KUKA KRL program: MyProgram_053().src

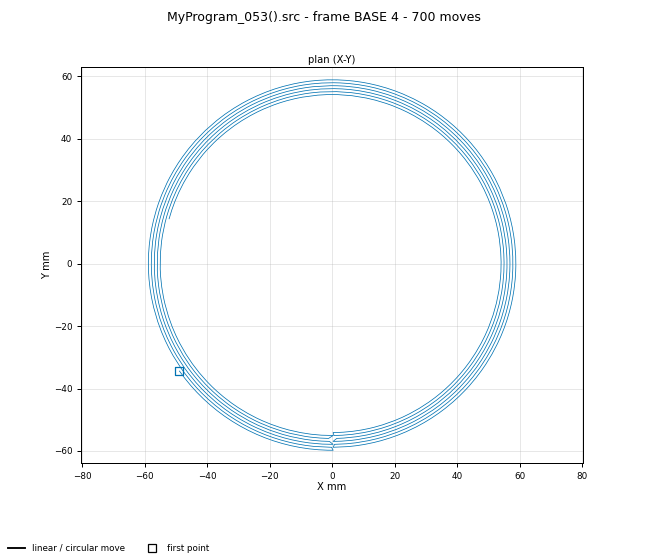
[picture p0: tool path of MyProgram_053().src in frame BASE 4, 700 of 700 moves have a stored position in this frame; points joined in program order, loops and branches not executed]
&ACCESS RVP
&REL 1
&PARAM TEMPLATE = C:\KRC\Roboter\Template\vorgabe
&PARAM EDITMASK = *
DEF MyProgram_053()
; ---- Setting reference (Base) ----
$BASE = BASE_DATA[4]

; --------------------------
; ---- Setting tool (TCP) ----
$TOOL = TOOL_DATA[3]
; --------------------------

$VEL.CP = VEL_APROX_PRINT
Startdeposition()
$VEL.CP = VEL_PRINT
LIN {X -48.8632,Y -34.4133,Z 68,A -149.9569,B 24.8869,C -2.4546,E1 24.8703,E2 233.9188} C_DIS
LIN {X -47.1157,Y -36.7695,Z 68,A -147.1292,B 24.8875,C -2.4482,E1 24.8751,E2 231.0929} C_DIS
LIN {X -45.2548,Y -39.0371,Z 68,A -144.3022,B 24.8881,C -2.4421,E1 24.8802,E2 228.2675} C_DIS
LIN {X -43.2848,Y -41.2106,Z 68,A -141.476,B 24.8886,C -2.4363,E1 24.8855,E2 225.4427} C_DIS
LIN {X -41.2106,Y -43.2848,Z 68,A -138.6504,B 24.8891,C -2.4308,E1 24.8912,E2 222.6185} C_DIS
LIN {X -39.0371,Y -45.2548,Z 68,A -135.8256,B 24.8896,C -2.4257,E1 24.8971,E2 219.7948} C_DIS
LIN {X -36.7695,Y -47.1157,Z 68,A -133.0016,B 24.89,C -2.4208,E1 24.9032,E2 216.9717} C_DIS
LIN {X -34.4133,Y -48.8632,Z 68,A -130.1785,B 24.8904,C -2.4164,E1 24.9096,E2 214.1495} C_DIS
LIN {X -31.9743,Y -50.4929,Z 68,A -127.3562,B 24.8908,C -2.4123,E1 24.9162,E2 211.3278} C_DIS
LIN {X -29.4582,Y -52.001,Z 68,A -124.535,B 24.8911,C -2.4085,E1 24.923,E2 208.5071} C_DIS
LIN {X -26.8711,Y -53.3838,Z 68,A -121.7145,B 24.8914,C -2.4052,E1 24.93,E2 205.6868} C_DIS
LIN {X -24.2194,Y -54.638,Z 68,A -118.8949,B 24.8917,C -2.4022,E1 24.9372,E2 202.8673} C_DIS
LIN {X -21.5092,Y -55.7606,Z 68,A -116.0763,B 24.8919,C -2.3996,E1 24.9445,E2 200.0486} C_DIS
LIN {X -18.7473,Y -56.7488,Z 68,A -113.2587,B 24.8921,C -2.3975,E1 24.9519,E2 197.2308} C_DIS
LIN {X -15.9402,Y -57.6003,Z 68,A -110.442,B 24.8923,C -2.3957,E1 24.9595,E2 194.4137} C_DIS
LIN {X -13.0946,Y -58.3131,Z 68,A -107.6262,B 24.8924,C -2.3943,E1 24.9672,E2 191.5974} C_DIS
LIN {X -10.2176,Y -58.8854,Z 68,A -104.8115,B 24.8925,C -2.3934,E1 24.9749,E2 188.7819} C_DIS
LIN {X -7.3159,Y -59.3158,Z 68,A -101.9978,B 24.8925,C -2.3929,E1 24.9827,E2 185.9674} C_DIS
LIN {X -4.3966,Y -59.6033,Z 68,A -99.185,B 24.8925,C -2.3928,E1 24.9905,E2 183.1534} C_DIS
LIN {X -1.4667,Y -59.7473,Z 68,A -96.3732,B 24.8925,C -2.3931,E1 24.9984,E2 180.3404} C_DIS
LIN {X 0.3491,Y -59.761,Z 68,A -94.9522,B 24.8931,C -2.3867,E1 25.0023,E2 178.9345} C_DIS
Enddeposition()
LIN {X 0.3491,Y -59.761,Z 68,A -94.9522,B 24.8931,C -2.3867,E1 25.0023,E2 178.9345} C_DIS
Startdeposition()
$VEL.CP = VEL_PRINT
LIN {X -0.1819,Y -58.8204,Z 68,A -97.1859,B 24.8948,C -2.3675,E1 24.9959,E2 181.214} C_DIS
LIN {X -5.9002,Y -58.5242,Z 68,A -102.0888,B 24.8936,C -2.3811,E1 24.9823,E2 186.0865} C_DIS
LIN {X -8.5559,Y -58.1955,Z 68,A -104.7263,B 24.8936,C -2.381,E1 24.975,E2 188.7262} C_DIS
LIN {X -11.2936,Y -57.7263,Z 68,A -107.3881,B 24.8935,C -2.3828,E1 24.9677,E2 191.3865} C_DIS
LIN {X -13.5936,Y -57.2291,Z 68,A -109.6463,B 24.8933,C -2.3845,E1 24.9616,E2 193.6434} C_DIS
LIN {X -16.2017,Y -56.5453,Z 68,A -112.2527,B 24.8931,C -2.3865,E1 24.9546,E2 196.2491} C_DIS
LIN {X -18.7885,Y -55.7389,Z 68,A -114.9287,B 24.8931,C -2.3878,E1 24.9475,E2 198.9269} C_DIS
LIN {X -21.2101,Y -54.8641,Z 68,A -117.4602,B 24.8928,C -2.3896,E1 24.9408,E2 201.4594} C_DIS
LIN {X -23.7558,Y -53.8105,Z 68,A -120.2317,B 24.8928,C -2.3907,E1 24.9337,E2 204.2348} C_DIS
LIN {X -25.9322,Y -52.7959,Z 68,A -122.5861,B 24.8925,C -2.3931,E1 24.9278,E2 206.5894} C_DIS
LIN {X -28.4573,Y -51.479,Z 68,A -125.2177,B 24.892,C -2.3994,E1 24.9213,E2 209.2134} C_DIS
LIN {X -30.7514,Y -50.1414,Z 68,A -127.767,B 24.8916,C -2.4038,E1 24.9152,E2 211.7601} C_DIS
LIN {X -32.928,Y -48.74,Z 68,A -130.3398,B 24.8913,C -2.4067,E1 24.9092,E2 214.3343} C_DIS
LIN {X -35.0695,Y -47.2236,Z 68,A -133.0589,B 24.8912,C -2.4079,E1 24.9031,E2 217.06} C_DIS
LIN {X -37.4099,Y -45.3916,Z 68,A -135.9134,B 24.8906,C -2.4139,E1 24.8968,E2 219.9109} C_DIS
LIN {X -39.5852,Y -43.5076,Z 68,A -138.9686,B 24.8906,C -2.4147,E1 24.8905,E2 222.9763} C_DIS
LIN {X -41.8366,Y -41.3466,Z 68,A -141.552,B 24.8892,C -2.4292,E1 24.8854,E2 225.536} C_DIS
LIN {X -43.5144,Y -39.5778,Z 68,A -144.139,B 24.8892,C -2.4305,E1 24.8804,E2 228.1313} C_DIS
LIN {X -45.2938,Y -37.5276,Z 68,A -146.7416,B 24.8885,C -2.4373,E1 24.8757,E2 230.7297} C_DIS
LIN {X -47.1481,Y -35.17,Z 68,A -149.431,B 24.8875,C -2.4483,E1 24.8712,E2 233.4055} C_DIS
LIN {X -48.4091,Y -33.4131,Z 68,A -151.8886,B 24.8875,C -2.4472,E1 24.8672,E2 235.8778} C_DIS
LIN {X -50.8588,Y -29.5512,Z 68,A -156.2944,B 24.8865,C -2.4595,E1 24.8607,E2 240.2766} C_DIS
LIN {X -52.1891,Y -27.1337,Z 68,A -159.076,B 24.886,C -2.4651,E1 24.857,E2 243.0598} C_DIS
LIN {X -53.4194,Y -24.6223,Z 68,A -161.8237,B 24.8853,C -2.4722,E1 24.8538,E2 245.8054} C_DIS
LIN {X -54.6088,Y -21.8592,Z 68,A -164.7604,B 24.8845,C -2.4803,E1 24.8506,E2 248.739} C_DIS
LIN {X -55.7868,Y -18.6465,Z 68,A -167.6273,B 24.8829,C -2.498,E1 24.8479,E2 251.5798} C_DIS
LIN {X -57.0985,Y -14.1292,Z 68,A -172.2395,B 24.8816,C -2.5111,E1 24.8444,E2 256.1874} C_DIS
LIN {X -57.7937,Y -10.9433,Z 68,A -175.929,B 24.8816,C -2.512,E1 24.8422,E2 259.8966} C_DIS
LIN {X -58.2622,Y -8.0862,Z 68,A -178.8137,B 24.8808,C -2.5196,E1 24.841,E2 262.7802} C_DIS
LIN {X -58.6196,Y -4.8584,Z 68,A 178.0495,B 24.8799,C -2.5299,E1 24.8402,E2 265.9112} C_DIS
LIN {X -58.7827,Y -2.13,Z 68,A 175.3754,B 24.8791,C -2.538,E1 24.8398,E2 268.582} C_DIS
LIN {X -58.82,Y 0.4129,Z 68,A 172.7179,B 24.8786,C -2.5428,E1 24.8398,E2 271.2441} C_DIS
LIN {X -58.7265,Y 3.3237,Z 68,A 170.0395,B 24.8775,C -2.5544,E1 24.8401,E2 273.9108} C_DIS
LIN {X -58.5256,Y 5.8861,Z 68,A 167.6002,B 24.8766,C -2.5634,E1 24.8408,E2 276.3433} C_DIS
LIN {X -58.2079,Y 8.4688,Z 68,A 164.903,B 24.8761,C -2.5687,E1 24.8418,E2 279.044} C_DIS
LIN {X -57.7129,Y 11.3629,Z 68,A 162.0961,B 24.8752,C -2.5785,E1 24.8432,E2 281.844} C_DIS
LIN {X -57.1771,Y 13.8072,Z 68,A 159.7574,B 24.8743,C -2.5878,E1 24.8446,E2 284.1743} C_DIS
LIN {X -56.2843,Y 17.0892,Z 68,A 156.5483,B 24.8731,C -2.5998,E1 24.847,E2 287.3733} C_DIS
LIN {X -55.6014,Y 19.1939,Z 68,A 154.0471,B 24.8731,C -2.6005,E1 24.8493,E2 289.8871} C_DIS
LIN {X -54.5799,Y 21.9303,Z 68,A 150.4175,B 24.8735,C -2.5959,E1 24.853,E2 293.5481} C_DIS
LIN {X -52.8589,Y 25.805,Z 68,A 147.4075,B 24.8704,C -2.6269,E1 24.8565,E2 296.5002} C_DIS
LIN {X -52.0364,Y 27.4235,Z 68,A 145.281,B 24.8705,C -2.6259,E1 24.8592,E2 298.6405} C_DIS
LIN {X -50.7407,Y 29.7534,Z 68,A 142.7868,B 24.8696,C -2.635,E1 24.8627,E2 301.1259} C_DIS
LIN {X -49.2458,Y 32.1676,Z 68,A 139.8519,B 24.8692,C -2.6398,E1 24.8671,E2 304.0643} C_DIS
LIN {X -47.8916,Y 34.1501,Z 68,A 137.5081,B 24.8685,C -2.646,E1 24.8708,E2 306.4049} C_DIS
LIN {X -45.9649,Y 36.7021,Z 68,A 134.4363,B 24.8676,C -2.6549,E1 24.8761,E2 309.47} C_DIS
LIN {X -43.8935,Y 39.1557,Z 68,A 130.9326,B 24.8676,C -2.6562,E1 24.8825,E2 312.9864} C_DIS
LIN {X -40.5775,Y 42.5843,Z 68,A 126.1334,B 24.8667,C -2.6645,E1 24.892,E2 317.7861} C_DIS
LIN {X -36.8982,Y 45.8082,Z 68,A 121.4315,B 24.8655,C -2.676,E1 24.902,E2 322.4785} C_DIS
LIN {X -34.2453,Y 47.8237,Z 68,A 118.3432,B 24.8646,C -2.6854,E1 24.909,E2 325.5554} C_DIS
LIN {X -31.4406,Y 49.7134,Z 68,A 115.1794,B 24.8637,C -2.6939,E1 24.9163,E2 328.7091} C_DIS
LIN {X -28.7227,Y 51.3307,Z 68,A 112.2925,B 24.8628,C -2.7029,E1 24.9233,E2 331.5834} C_DIS
LIN {X -26.8061,Y 52.3571,Z 68,A 109.9748,B 24.8628,C -2.7027,E1 24.929,E2 333.9079} C_DIS
LIN {X -24.1417,Y 53.6378,Z 68,A 106.9814,B 24.8626,C -2.7049,E1 24.9366,E2 336.9034} C_DIS
LIN {X -21.1328,Y 54.894,Z 68,A 103.9362,B 24.8619,C -2.7116,E1 24.9445,E2 339.9394} C_DIS
LIN {X -18.4448,Y 55.8547,Z 68,A 101.1212,B 24.8616,C -2.7143,E1 24.9519,E2 342.7533} C_DIS
LIN {X -15.7595,Y 56.6706,Z 68,A 98.3718,B 24.8614,C -2.7169,E1 24.9593,E2 345.5009} C_DIS
LIN {X -12.2609,Y 57.529,Z 68,A 95.0311,B 24.8607,C -2.7233,E1 24.9683,E2 348.8308} C_DIS
LIN {X -9.8349,Y 57.9925,Z 68,A 92.5949,B 24.8606,C -2.7246,E1 24.975,E2 351.2667} C_DIS
LIN {X -7.116,Y 58.389,Z 68,A 89.8714,B 24.8606,C -2.7253,E1 24.9826,E2 353.9905} C_DIS
LIN {X -4.5936,Y 58.6408,Z 68,A 87.3044,B 24.8606,C -2.7246,E1 24.9897,E2 356.5605} C_DIS
LIN {X -1.5185,Y 58.8015,Z 68,A 84.2474,B 24.8606,C -2.7244,E1 24.9982,E2 359.6185} C_DIS
LIN {X 1.6458,Y 58.7976,Z 68,A 81.222,B 24.8604,C -2.726,E1 25.0067,E2 362.6398} C_DIS
LIN {X 4.5596,Y 58.6435,Z 68,A 78.5253,B 24.8601,C -2.7289,E1 25.0142,E2 365.3284} C_DIS
LIN {X 7.0083,Y 58.4016,Z 68,A 76.0735,B 24.8603,C -2.7274,E1 25.021,E2 367.782} C_DIS
LIN {X 9.7413,Y 58.0082,Z 68,A 73.563,B 24.86,C -2.7303,E1 25.0279,E2 370.2833} C_DIS
LIN {X 11.8943,Y 57.6053,Z 68,A 71.2881,B 24.8604,C -2.7265,E1 25.0341,E2 372.5645} C_DIS
LIN {X 14.4994,Y 57.0055,Z 68,A 68.5573,B 24.8608,C -2.7225,E1 25.0416,E2 375.3009} C_DIS
LIN {X 17.4989,Y 56.1572,Z 68,A 65.5349,B 24.861,C -2.7206,E1 25.0496,E2 378.3225} C_DIS
LIN {X 20.1878,Y 55.2475,Z 68,A 62.629,B 24.8615,C -2.7153,E1 25.0573,E2 381.2352} C_DIS
LIN {X 22.6593,Y 54.2811,Z 68,A 59.8471,B 24.8622,C -2.7085,E1 25.0645,E2 384.0268} C_DIS
LIN {X 26.0847,Y 52.7203,Z 68,A 56.5042,B 24.862,C -2.7111,E1 25.0729,E2 387.3549} C_DIS
LIN {X 29.0426,Y 51.1513,Z 68,A 53.5864,B 24.8617,C -2.7141,E1 25.08,E2 390.2571} C_DIS
LIN {X 30.8083,Y 50.1077,Z 68,A 51.3127,B 24.8626,C -2.7052,E1 25.0855,E2 392.5448} C_DIS
LIN {X 32.9546,Y 48.722,Z 68,A 49.0436,B 24.8625,C -2.7061,E1 25.0908,E2 394.8043} C_DIS
LIN {X 34.8992,Y 47.3489,Z 68,A 46.4804,B 24.8634,C -2.6968,E1 25.0966,E2 397.3804} C_DIS
LIN {X 37.2606,Y 45.5144,Z 68,A 43.5291,B 24.864,C -2.6907,E1 25.1031,E2 400.3352} C_DIS
LIN {X 39.066,Y 43.9743,Z 68,A 41.4039,B 24.864,C -2.6904,E1 25.1075,E2 402.4528} C_DIS
LIN {X 41.0256,Y 42.1523,Z 68,A 38.6909,B 24.8648,C -2.6827,E1 25.113,E2 405.1728} C_DIS
LIN {X 42.9045,Y 40.2373,Z 68,A 36.1779,B 24.8652,C -2.6794,E1 25.1179,E2 407.6827} C_DIS
LIN {X 44.4749,Y 38.4953,Z 68,A 33.8185,B 24.8659,C -2.6726,E1 25.1222,E2 410.0477} C_DIS
LIN {X 46.2369,Y 36.3594,Z 68,A 31.1846,B 24.8664,C -2.6678,E1 25.1268,E2 412.6808} C_DIS
LIN {X 47.8292,Y 34.2376,Z 68,A 28.6547,B 24.8669,C -2.6627,E1 25.131,E2 415.2104} C_DIS
LIN {X 49.4968,Y 31.7789,Z 68,A 25.6809,B 24.8678,C -2.6536,E1 25.1356,E2 418.1909} C_DIS
LIN {X 51.014,Y 29.2815,Z 68,A 22.9579,B 24.8682,C -2.649,E1 25.1395,E2 420.9109} C_DIS
LIN {X 52.2323,Y 27.0503,Z 68,A 19.8319,B 24.8704,C -2.6275,E1 25.1436,E2 424.0712} C_DIS
LIN {X 53.6588,Y 24.0952,Z 68,A 16.7232,B 24.8711,C -2.6206,E1 25.1472,E2 427.1794} C_DIS
LIN {X 55.5872,Y 19.2344,Z 68,A 12.4414,B 24.8707,C -2.6247,E1 25.1514,E2 431.4277} C_DIS
LIN {X 56.2835,Y 17.0915,Z 68,A 9.9975,B 24.8719,C -2.6124,E1 25.1535,E2 433.8867} C_DIS
LIN {X 57.0667,Y 14.2598,Z 68,A 7.2199,B 24.8725,C -2.6058,E1 25.1554,E2 436.6639} C_DIS
LIN {X 57.6695,Y 11.5813,Z 68,A 4.5156,B 24.8734,C -2.597,E1 25.157,E2 439.3734} C_DIS
LIN {X 58.1359,Y 8.9473,Z 68,A 1.9962,B 24.874,C -2.591,E1 25.1582,E2 441.8921} C_DIS
LIN {X 58.4681,Y 6.4352,Z 68,A -0.6025,B 24.875,C -2.5803,E1 25.159,E2 444.5008} C_DIS
LIN {X 58.7635,Y 2.5865,Z 68,A -4.6079,B 24.8767,C -2.5628,E1 25.1597,E2 448.5238} C_DIS
LIN {X 58.8186,Y -0.5568,Z 68,A -7.0159,B 24.8762,C -2.5684,E1 25.1597,E2 450.9042} C_DIS
LIN {X 58.7666,Y -2.5145,Z 68,A -9.2638,B 24.8775,C -2.5544,E1 25.1595,E2 453.1719} C_DIS
LIN {X 58.6012,Y -5.0835,Z 68,A -11.8045,B 24.8783,C -2.5457,E1 25.159,E2 455.718} C_DIS
LIN {X 58.2064,Y -8.479,Z 68,A -14.7537,B 24.8785,C -2.5441,E1 25.1579,E2 458.6535} C_DIS
LIN {X 57.7979,Y -10.9214,Z 68,A -17.1892,B 24.8793,C -2.536,E1 25.1568,E2 461.094} C_DIS
LIN {X 57.378,Y -12.9497,Z 68,A -19.3393,B 24.8802,C -2.5265,E1 25.1555,E2 463.2539} C_DIS
LIN {X 56.7813,Y -15.3532,Z 68,A -21.7826,B 24.881,C -2.5183,E1 25.1538,E2 465.7025} C_DIS
LIN {X 55.9859,Y -18.0394,Z 68,A -24.5467,B 24.8818,C -2.5091,E1 25.1515,E2 468.4728} C_DIS
LIN {X 55.1025,Y -20.5821,Z 68,A -27.008,B 24.8822,C -2.5049,E1 25.1492,E2 470.9302} C_DIS
LIN {X 54.1298,Y -23.0182,Z 68,A -29.6221,B 24.8831,C -2.4958,E1 25.1464,E2 473.5513} C_DIS
LIN {X 52.9555,Y -25.6042,Z 68,A -32.7817,B 24.8847,C -2.4785,E1 25.1426,E2 476.7347} C_DIS
LIN {X 51.1574,Y -29.0321,Z 68,A -36.2551,B 24.8851,C -2.4745,E1 25.1379,E2 480.1994} C_DIS
LIN {X 49.1785,Y -32.2697,Z 68,A -39.6052,B 24.8853,C -2.4722,E1 25.133,E2 483.5379} C_DIS
LIN {X 47.8134,Y -34.2598,Z 68,A -42.1617,B 24.8863,C -2.4611,E1 25.1289,E2 486.1083} C_DIS
LIN {X 46.0279,Y -36.6239,Z 68,A -45.2761,B 24.8875,C -2.4483,E1 25.1235,E2 489.2384} C_DIS
LIN {X 43.9528,Y -39.09,Z 68,A -47.6687,B 24.8867,C -2.4574,E1 25.1192,E2 491.5985} C_DIS
LIN {X 42.6761,Y -40.4803,Z 68,A -49.9852,B 24.8881,C -2.442,E1 25.1148,E2 493.9414} C_DIS
LIN {X 40.7579,Y -42.4104,Z 68,A -52.5538,B 24.8885,C -2.4375,E1 25.1096,E2 496.5096} C_DIS
LIN {X 38.7295,Y -44.2704,Z 68,A -55.3493,B 24.8893,C -2.4288,E1 25.1038,E2 499.3146} C_DIS
LIN {X 36.2424,Y -46.3294,Z 68,A -58.2487,B 24.8894,C -2.4276,E1 25.0975,E2 502.2061} C_DIS
LIN {X 34.2378,Y -47.829,Z 68,A -60.8411,B 24.8902,C -2.4191,E1 25.0917,E2 504.8092} C_DIS
LIN {X 31.8563,Y -49.4472,Z 68,A -63.6213,B 24.8906,C -2.4143,E1 25.0852,E2 507.5917} C_DIS
LIN {X 29.4736,Y -50.9037,Z 68,A -66.3447,B 24.8911,C -2.4093,E1 25.0786,E2 510.3185} C_DIS
LIN {X 26.9019,Y -52.3082,Z 68,A -69.5131,B 24.8921,C -2.3976,E1 25.0708,E2 513.5057} C_DIS
LIN {X 23.6635,Y -53.8508,Z 68,A -72.6989,B 24.892,C -2.399,E1 25.0627,E2 516.6802} C_DIS
LIN {X 21.0515,Y -54.9247,Z 68,A -75.3162,B 24.892,C -2.3981,E1 25.0559,E2 519.2936} C_DIS
LIN {X 18.5531,Y -55.8175,Z 68,A -77.9819,B 24.8925,C -2.3931,E1 25.0489,E2 521.9659} C_DIS
LIN {X 15.6483,Y -56.7016,Z 68,A -80.8451,B 24.8926,C -2.3919,E1 25.0412,E2 524.8271} C_DIS
LIN {X 13.3649,Y -57.2821,Z 68,A -83.2555,B 24.8931,C -2.3872,E1 25.0346,E2 527.2451} C_DIS
LIN {X 10.4333,Y -57.8877,Z 68,A -86.3232,B 24.8936,C -2.3816,E1 25.0262,E2 530.3225} C_DIS
LIN {X 7.9324,Y -58.2841,Z 68,A -88.6588,B 24.8935,C -2.3827,E1 25.0198,E2 532.6536} C_DIS
LIN {X 5.1225,Y -58.5975,Z 68,A -91.9162,B 24.8945,C -2.3708,E1 25.0106,E2 535.9372} C_DIS
LIN {X 0.3303,Y -58.8102,Z 68,A -94.5805,B 24.8909,C -2.4111,E1 25.0035,E2 538.505} C_DIS
Enddeposition()
LIN {X 0.3303,Y -58.8102,Z 68,A -94.5805,B 24.8909,C -2.4111,E1 25.0035,E2 538.505} C_DIS
Startdeposition()
$VEL.CP = VEL_PRINT
LIN {X 0.78,Y -57.8714,Z 68,A -94.0127,B 24.8892,C -2.4297,E1 25.0052,E2 537.8931} C_DIS
LIN {X 4.6739,Y -57.6876,Z 68,A -90.3787,B 24.8895,C -2.4267,E1 25.0153,E2 534.2679} C_DIS
LIN {X 7.6047,Y -57.3751,Z 68,A -87.8197,B 24.89,C -2.4209,E1 25.0223,E2 531.7245} C_DIS
LIN {X 11.7052,Y -56.6807,Z 68,A -83.3977,B 24.8891,C -2.4305,E1 25.0346,E2 527.2844} C_DIS
LIN {X 14.3445,Y -56.0709,Z 68,A -80.677,B 24.8888,C -2.434,E1 25.0419,E2 524.5596} C_DIS
LIN {X 16.8623,Y -55.3665,Z 68,A -77.3217,B 24.887,C -2.4535,E1 25.051,E2 521.1637} C_DIS
LIN {X 20.8071,Y -54.0081,Z 68,A -74.1057,B 24.8884,C -2.4389,E1 25.0593,E2 517.9892} C_DIS
LIN {X 23.7341,Y -52.7864,Z 68,A -71.0499,B 24.8881,C -2.4416,E1 25.0672,E2 514.9342} C_DIS
LIN {X 26.6333,Y -51.3855,Z 68,A -67.275,B 24.8864,C -2.4598,E1 25.0767,E2 511.1266} C_DIS
LIN {X 29.9387,Y -49.5318,Z 68,A -63.9811,B 24.8868,C -2.4562,E1 25.0846,E2 507.8509} C_DIS
LIN {X 32.2718,Y -48.0446,Z 68,A -61.2572,B 24.8863,C -2.4611,E1 25.0909,E2 505.1244} C_DIS
LIN {X 34.2385,Y -46.663,Z 68,A -58.3006,B 24.8846,C -2.4791,E1 25.0977,E2 502.1358} C_DIS
LIN {X 37.217,Y -44.3246,Z 68,A -54.7007,B 24.8842,C -2.4838,E1 25.1055,E2 498.5384} C_DIS
LIN {X 39.9475,Y -41.8807,Z 68,A -51.5822,B 24.8845,C -2.4805,E1 25.1118,E2 495.4403} C_DIS
LIN {X 41.9102,Y -39.9168,Z 68,A -49.1055,B 24.8845,C -2.4809,E1 25.1166,E2 492.9733} C_DIS
LIN {X 43.3694,Y -38.325,Z 68,A -46.807,B 24.8836,C -2.49,E1 25.1209,E2 490.6637} C_DIS
LIN {X 45.094,Y -36.2803,Z 68,A -43.6872,B 24.882,C -2.5077,E1 25.1265,E2 487.5162} C_DIS
LIN {X 47.3207,Y -33.3254,Z 68,A -40.5794,B 24.8822,C -2.5046,E1 25.1316,E2 484.4308} C_DIS
LIN {X 49.4641,Y -30.0499,Z 68,A -36.7413,B 24.8813,C -2.5145,E1 25.1374,E2 480.5885} C_DIS
LIN {X 51.079,Y -27.2161,Z 68,A -33.062,B 24.8794,C -2.5343,E1 25.1424,E2 476.8817} C_DIS
LIN {X 52.4942,Y -24.3734,Z 68,A -29.8313,B 24.8784,C -2.5456,E1 25.1463,E2 473.6416} C_DIS
LIN {X 53.9012,Y -21.0802,Z 68,A -26.7204,B 24.8784,C -2.546,E1 25.1495,E2 470.5469} C_DIS
LIN {X 54.8699,Y -18.412,Z 68,A -23.9576,B 24.8776,C -2.5535,E1 25.1521,E2 467.782} C_DIS
LIN {X 55.6901,Y -15.7582,Z 68,A -21.1575,B 24.8767,C -2.5632,E1 25.1543,E2 464.975} C_DIS
LIN {X 56.3798,Y -13.0776,Z 68,A -18.2243,B 24.8754,C -2.5763,E1 25.1562,E2 462.0278} C_DIS
LIN {X 57.06,Y -9.6894,Z 68,A -15.5141,B 24.876,C -2.5703,E1 25.1576,E2 459.3477} C_DIS
LIN {X 57.3952,Y -7.4494,Z 68,A -12.8681,B 24.8744,C -2.5868,E1 25.1587,E2 456.6781} C_DIS
LIN {X 57.6691,Y -4.9056,Z 68,A -10.2228,B 24.8733,C -2.5975,E1 25.1594,E2 454.0233} C_DIS
LIN {X 57.8559,Y -1.5642,Z 68,A -7.0469,B 24.8726,C -2.6047,E1 25.1598,E2 450.8492} C_DIS
LIN {X 57.835,Y 2.208,Z 68,A -2.7929,B 24.8702,C -2.6287,E1 25.1595,E2 446.5637} C_DIS
LIN {X 57.5655,Y 5.9934,Z 68,A 0.3996,B 24.8704,C -2.6272,E1 25.1587,E2 443.3939} C_DIS
LIN {X 57.306,Y 8.1072,Z 68,A 2.4235,B 24.87,C -2.6317,E1 25.158,E2 441.3712} C_DIS
LIN {X 56.8276,Y 10.9692,Z 68,A 5.2758,B 24.8691,C -2.64,E1 25.1566,E2 438.5158} C_DIS
LIN {X 56.281,Y 13.4982,Z 68,A 7.9804,B 24.868,C -2.6511,E1 25.1549,E2 435.8006} C_DIS
LIN {X 55.5222,Y 16.3404,Z 68,A 11.1766,B 24.8665,C -2.6665,E1 25.1524,E2 432.5866} C_DIS
LIN {X 54.66,Y 19.0265,Z 68,A 13.9132,B 24.8658,C -2.6733,E1 25.1499,E2 429.8492} C_DIS
LIN {X 53.2238,Y 22.7362,Z 68,A 17.4466,B 24.8656,C -2.6751,E1 25.1462,E2 426.3311} C_DIS
LIN {X 52.3711,Y 24.6379,Z 68,A 19.8863,B 24.8642,C -2.6895,E1 25.1433,E2 423.8704} C_DIS
LIN {X 50.7121,Y 27.8945,Z 68,A 23.1418,B 24.864,C -2.6908,E1 25.1391,E2 420.629} C_DIS
LIN {X 49.2661,Y 30.3755,Z 68,A 25.9891,B 24.8633,C -2.6983,E1 25.135,E2 417.7785} C_DIS
LIN {X 46.9666,Y 33.8217,Z 68,A 30.0766,B 24.8623,C -2.7082,E1 25.1285,E2 413.6878} C_DIS
LIN {X 45.1647,Y 36.1933,Z 68,A 32.9551,B 24.8617,C -2.7136,E1 25.1236,E2 410.8102} C_DIS
LIN {X 42.987,Y 38.7539,Z 68,A 36.4163,B 24.8606,C -2.724,E1 25.1172,E2 407.3397} C_DIS
LIN {X 40.9213,Y 40.9299,Z 68,A 39.2019,B 24.8604,C -2.7262,E1 25.1118,E2 404.561} C_DIS
LIN {X 38.9759,Y 42.7858,Z 68,A 42.0048,B 24.8595,C -2.7346,E1 25.1061,E2 401.7494} C_DIS
LIN {X 35.9351,Y 45.3693,Z 68,A 45.8643,B 24.859,C -2.7399,E1 25.0977,E2 397.8922} C_DIS
LIN {X 33.3247,Y 47.3211,Z 68,A 49.4908,B 24.8575,C -2.7541,E1 25.0895,E2 394.2447} C_DIS
LIN {X 30.0673,Y 49.4536,Z 68,A 52.826,B 24.8581,C -2.7487,E1 25.0817,E2 390.9332} C_DIS
LIN {X 28.3743,Y 50.4444,Z 68,A 54.9276,B 24.8575,C -2.7548,E1 25.0765,E2 388.8234} C_DIS
LIN {X 25.8658,Y 51.7755,Z 68,A 57.6285,B 24.8573,C -2.756,E1 25.0698,E2 386.1271} C_DIS
LIN {X 23.1034,Y 53.0654,Z 68,A 60.6915,B 24.8569,C -2.7603,E1 25.062,E2 383.0614} C_DIS
LIN {X 19.916,Y 54.3417,Z 68,A 64.0369,B 24.8567,C -2.7624,E1 25.0533,E2 379.7183} C_DIS
LIN {X 17.1237,Y 55.2855,Z 68,A 67.2148,B 24.8559,C -2.7701,E1 25.0449,E2 376.528} C_DIS
LIN {X 13.9518,Y 56.1703,Z 68,A 70.152,B 24.8564,C -2.7654,E1 25.037,E2 373.6067} C_DIS
LIN {X 11.4099,Y 56.7413,Z 68,A 72.7812,B 24.8561,C -2.7676,E1 25.0298,E2 370.9756} C_DIS
LIN {X 8.4584,Y 57.2558,Z 68,A 75.9579,B 24.8556,C -2.7728,E1 25.021,E2 367.7895} C_DIS
LIN {X 5.2145,Y 57.6413,Z 68,A 78.8815,B 24.8562,C -2.767,E1 25.0129,E2 364.8818} C_DIS
LIN {X 2.545,Y 57.8207,Z 68,A 81.3542,B 24.8566,C -2.7634,E1 25.0061,E2 362.4185} C_DIS
LIN {X 0.4353,Y 57.875,Z 68,A 83.7312,B 24.856,C -2.7688,E1 24.9994,E2 360.0289} C_DIS
LIN {X -3.3089,Y 57.7821,Z 68,A 87.6438,B 24.8557,C -2.7717,E1 24.9884,E2 356.1087} C_DIS
LIN {X -6.6039,Y 57.4988,Z 68,A 90.5962,B 24.8565,C -2.7638,E1 24.9803,E2 353.1736} C_DIS
LIN {X -9.1846,Y 57.1442,Z 68,A 93.2568,B 24.8565,C -2.7636,E1 24.9729,E2 350.5111} C_DIS
LIN {X -11.1973,Y 56.7837,Z 68,A 95.4579,B 24.8564,C -2.7655,E1 24.9669,E2 348.3032} C_DIS
LIN {X -14.0822,Y 56.1382,Z 68,A 98.1948,B 24.857,C -2.7591,E1 24.9595,E2 345.5776} C_DIS
LIN {X -16.899,Y 55.3551,Z 68,A 101.1648,B 24.8572,C -2.7575,E1 24.9515,E2 342.6067} C_DIS
LIN {X -19.5753,Y 54.4664,Z 68,A 103.8788,B 24.8577,C -2.7526,E1 24.9444,E2 339.8991} C_DIS
LIN {X -22.3538,Y 53.3856,Z 68,A 106.9839,B 24.8578,C -2.7515,E1 24.9363,E2 336.7897} C_DIS
LIN {X -25.3527,Y 52.0293,Z 68,A 110.1218,B 24.8585,C -2.7443,E1 24.9284,E2 333.6611} C_DIS
LIN {X -27.4671,Y 50.944,Z 68,A 113.0058,B 24.8579,C -2.7503,E1 24.9212,E2 330.7548} C_DIS
LIN {X -30.3801,Y 49.2631,Z 68,A 115.7209,B 24.8597,C -2.7331,E1 24.9148,E2 328.0726} C_DIS
LIN {X -32.9008,Y 47.6158,Z 68,A 118.8661,B 24.86,C -2.7303,E1 24.9075,E2 324.9234} C_DIS
LIN {X -34.952,Y 46.131,Z 68,A 121.649,B 24.86,C -2.7303,E1 24.9013,E2 322.1309} C_DIS
LIN {X -38.0309,Y 43.6274,Z 68,A 125.0474,B 24.8618,C -2.7122,E1 24.894,E2 318.7624} C_DIS
LIN {X -39.9503,Y 41.878,Z 68,A 128.078,B 24.8616,C -2.7145,E1 24.8878,E2 315.7141} C_DIS
LIN {X -41.6921,Y 40.1432,Z 68,A 130.066,B 24.863,C -2.7008,E1 24.884,E2 313.7502} C_DIS
LIN {X -43.2066,Y 38.5086,Z 68,A 132.5738,B 24.863,C -2.7007,E1 24.8792,E2 311.2317} C_DIS
LIN {X -44.8223,Y 36.6158,Z 68,A 134.9729,B 24.8638,C -2.6933,E1 24.875,E2 308.8392} C_DIS
LIN {X -46.7908,Y 34.0639,Z 68,A 138.0557,B 24.8648,C -2.683,E1 24.8698,E2 305.7661} C_DIS
LIN {X -48.0905,Y 32.2039,Z 68,A 140.8524,B 24.8645,C -2.6864,E1 24.8654,E2 302.9474} C_DIS
LIN {X -49.9727,Y 29.1979,Z 68,A 144.0823,B 24.866,C -2.6717,E1 24.8607,E2 299.736} C_DIS
LIN {X -51.3637,Y 26.6755,Z 68,A 146.8569,B 24.8669,C -2.6622,E1 24.8571,E2 296.9694} C_DIS
LIN {X -52.8218,Y 23.6552,Z 68,A 150.0844,B 24.868,C -2.6509,E1 24.8533,E2 293.7513} C_DIS
LIN {X -53.6201,Y 21.785,Z 68,A 152.3867,B 24.8682,C -2.6498,E1 24.8508,E2 291.4388} C_DIS
LIN {X -54.7886,Y 18.6532,Z 68,A 155.5045,B 24.8695,C -2.6365,E1 24.8479,E2 288.3352} C_DIS
LIN {X -55.3682,Y 16.8536,Z 68,A 158.1009,B 24.8688,C -2.6432,E1 24.8457,E2 285.7079} C_DIS
LIN {X -56.4794,Y 12.6446,Z 68,A 161.8983,B 24.871,C -2.621,E1 24.8432,E2 281.9414} C_DIS
LIN {X -57.0063,Y 10.0022,Z 68,A 164.5573,B 24.8719,C -2.6125,E1 24.8419,E2 279.2869} C_DIS
LIN {X -57.4397,Y 7.1061,Z 68,A 167.4696,B 24.8727,C -2.6036,E1 24.8408,E2 276.3785} C_DIS
LIN {X -57.7841,Y 3.272,Z 68,A 171.0504,B 24.8743,C -2.5877,E1 24.84,E2 272.8142} C_DIS
LIN {X -57.876,Y -0.4305,Z 68,A 175.0736,B 24.8748,C -2.5822,E1 24.8398,E2 268.78} C_DIS
LIN {X -57.7878,Y -3.2048,Z 68,A 177.7218,B 24.8758,C -2.5719,E1 24.8401,E2 266.1406} C_DIS
LIN {X -57.4786,Y -6.776,Z 68,A -178.1855,B 24.876,C -2.5701,E1 24.8413,E2 262.0275} C_DIS
LIN {X -56.8854,Y -10.6693,Z 68,A -174.7203,B 24.8779,C -2.5507,E1 24.8429,E2 258.5881} C_DIS
LIN {X -56.3281,Y -13.3014,Z 68,A -171.1865,B 24.8772,C -2.5577,E1 24.8452,E2 255.0169} C_DIS
LIN {X -55.1745,Y -17.4811,Z 68,A -167.1306,B 24.8788,C -2.5409,E1 24.8485,E2 250.9778} C_DIS
LIN {X -53.8888,Y -21.1118,Z 68,A -164.0836,B 24.8811,C -2.5166,E1 24.8514,E2 247.9717} C_DIS
LIN {X -52.8045,Y -23.6939,Z 68,A -161.0594,B 24.8814,C -2.5132,E1 24.8548,E2 244.9389} C_DIS
LIN {X -51.5463,Y -26.3188,Z 68,A -158.1799,B 24.8822,C -2.5053,E1 24.8583,E2 242.0627} C_DIS
LIN {X -50.6502,Y -28.0057,Z 68,A -156.3925,B 24.8828,C -2.4984,E1 24.8607,E2 240.2823} C_DIS
LIN {X -49.7083,Y -29.6449,Z 68,A -154.0153,B 24.8824,C -2.5025,E1 24.8641,E2 237.883} C_DIS
LIN {X -47.1531,Y -33.5603,Z 68,A -150.0117,B 24.8846,C -2.4799,E1 24.8703,E2 233.9136} C_DIS
LIN {X -45.9103,Y -35.2414,Z 68,A -147.539,B 24.8844,C -2.4821,E1 24.8745,E2 231.4237} C_DIS
LIN {X -43.5847,Y -38.0799,Z 68,A -144.0307,B 24.8853,C -2.4716,E1 24.8808,E2 227.9243} C_DIS
LIN {X -41.6382,Y -40.1991,Z 68,A -141.1778,B 24.8859,C -2.4656,E1 24.8863,E2 225.0734} C_DIS
LIN {X -39.9557,Y -41.8728,Z 68,A -138.6526,B 24.886,C -2.464,E1 24.8913,E2 222.5414} C_DIS
LIN {X -37.1147,Y -44.4098,Z 68,A -135.5205,B 24.8878,C -2.4451,E1 24.8979,E2 219.4421} C_DIS
LIN {X -34.303,Y -46.6157,Z 68,A -131.4108,B 24.8874,C -2.4495,E1 24.907,E2 215.307} C_DIS
LIN {X -32.0434,Y -48.1973,Z 68,A -128.7427,B 24.8879,C -2.444,E1 24.9131,E2 212.6431} C_DIS
LIN {X -29.2489,Y -49.9417,Z 68,A -125.3329,B 24.8881,C -2.4421,E1 24.9213,E2 209.2272} C_DIS
LIN {X -26.2122,Y -51.6008,Z 68,A -122.1193,B 24.8888,C -2.4337,E1 24.9292,E2 206.0248} C_DIS
LIN {X -24.455,Y -52.4562,Z 68,A -119.7543,B 24.8883,C -2.4398,E1 24.9352,E2 203.6393} C_DIS
LIN {X -21.2149,Y -53.8482,Z 68,A -116.5985,B 24.8892,C -2.4298,E1 24.9433,E2 200.5002} C_DIS
LIN {X -18.1455,Y -54.9595,Z 68,A -113.2706,B 24.8892,C -2.429,E1 24.9521,E2 197.1677} C_DIS
LIN {X -15.2826,Y -55.8228,Z 68,A -110.3222,B 24.8895,C -2.4268,E1 24.96,E2 194.2197} C_DIS
LIN {X -12.8848,Y -56.4243,Z 68,A -107.8951,B 24.8896,C -2.4252,E1 24.9666,E2 191.7931} C_DIS
LIN {X -9.7967,Y -57.042,Z 68,A -104.8882,B 24.8899,C -2.4219,E1 24.9749,E2 188.791} C_DIS
LIN {X -7.2781,Y -57.4174,Z 68,A -102.2579,B 24.8898,C -2.4236,E1 24.9822,E2 186.1546} C_DIS
LIN {X -3.1822,Y -57.7891,Z 68,A -97.8455,B 24.8891,C -2.4305,E1 24.9945,E2 181.724} C_DIS
LIN {X 0.3229,Y -57.875,Z 68,A -95.2638,B 24.8907,C -2.4129,E1 25.0016,E2 179.184} C_DIS
Enddeposition()
LIN {X 0.3229,Y -57.875,Z 68,A -95.2638,B 24.8907,C -2.4129,E1 25.0016,E2 179.184} C_DIS
Startdeposition()
$VEL.CP = VEL_PRINT
LIN {X -0.8687,Y -56.9265,Z 68,A -97.0968,B 24.8904,C -2.4162,E1 24.9965,E2 181.009} C_DIS
LIN {X -3.413,Y -56.8303,Z 68,A -100.1238,B 24.8913,C -2.4069,E1 24.988,E2 184.0589} C_DIS
LIN {X -6.1872,Y -56.5963,Z 68,A -102.6551,B 24.8908,C -2.4124,E1 24.981,E2 186.5786} C_DIS
LIN {X -8.8492,Y -56.2411,Z 68,A -105.738,B 24.8914,C -2.4057,E1 24.9724,E2 189.6799} C_DIS
LIN {X -13.1394,Y -55.3969,Z 68,A -109.7563,B 24.8906,C -2.4149,E1 24.9615,E2 193.6813} C_DIS
LIN {X -15.893,Y -54.6705,Z 68,A -112.596,B 24.8903,C -2.4172,E1 24.9538,E2 196.52} C_DIS
LIN {X -19.8657,Y -53.3555,Z 68,A -116.5403,B 24.8896,C -2.4256,E1 24.9435,E2 200.4518} C_DIS
LIN {X -23.7377,Y -51.7486,Z 68,A -121.0098,B 24.8896,C -2.4253,E1 24.932,E2 204.9324} C_DIS
LIN {X -26.4955,Y -50.3919,Z 68,A -124.1857,B 24.8894,C -2.4275,E1 24.924,E2 208.1114} C_DIS
LIN {X -30.2362,Y -48.2403,Z 68,A -128.3817,B 24.8886,C -2.4363,E1 24.9139,E2 212.2992} C_DIS
LIN {X -32.2209,Y -46.9391,Z 68,A -131.0775,B 24.8888,C -2.4345,E1 24.9077,E2 215.0082} C_DIS
LIN {X -35.3697,Y -44.6133,Z 68,A -134.7034,B 24.8876,C -2.4469,E1 24.8996,E2 218.6176} C_DIS
LIN {X -36.6303,Y -43.585,Z 68,A -136.6609,B 24.8879,C -2.4443,E1 24.8954,E2 220.5889} C_DIS
LIN {X -38.9639,Y -41.5111,Z 68,A -139.6225,B 24.887,C -2.4536,E1 24.8893,E2 223.5403} C_DIS
LIN {X -41.3962,Y -39.086,Z 68,A -142.6083,B 24.8856,C -2.469,E1 24.8835,E2 226.5019} C_DIS
LIN {X -43.226,Y -37.0526,Z 68,A -145.7654,B 24.8856,C -2.4681,E1 24.8776,E2 229.6754} C_DIS
LIN {X -44.7258,Y -35.2273,Z 68,A -148.3707,B 24.8856,C -2.4697,E1 24.873,E2 232.289} C_DIS
LIN {X -46.1011,Y -33.4083,Z 68,A -151.0577,B 24.8856,C -2.4686,E1 24.8686,E2 234.9917} C_DIS
LIN {X -47.9851,Y -30.6399,Z 68,A -153.8572,B 24.8839,C -2.4866,E1 24.8643,E2 237.7621} C_DIS
LIN {X -49.217,Y -28.6189,Z 68,A -156.4904,B 24.8838,C -2.4886,E1 24.8605,E2 240.4042} C_DIS
LIN {X -50.3046,Y -26.6612,Z 68,A -158.695,B 24.8831,C -2.4954,E1 24.8576,E2 242.6041} C_DIS
LIN {X -51.5741,Y -24.1137,Z 68,A -162.0829,B 24.8831,C -2.4946,E1 24.8535,E2 246.0124} C_DIS
LIN {X -53.1672,Y -20.3628,Z 68,A -165.5484,B 24.8811,C -2.5167,E1 24.8499,E2 249.4443} C_DIS
LIN {X -53.9562,Y -18.1681,Z 68,A -167.8047,B 24.8803,C -2.5251,E1 24.8478,E2 251.6936} C_DIS
LIN {X -54.7339,Y -15.6707,Z 68,A -170.9145,B 24.8803,C -2.5251,E1 24.8453,E2 254.8215} C_DIS
LIN {X -55.552,Y -12.4675,Z 68,A -173.7214,B 24.8786,C -2.5435,E1 24.8435,E2 257.6005} C_DIS
LIN {X -56.2783,Y -8.6076,Z 68,A -178.1213,B 24.8781,C -2.5483,E1 24.8413,E2 262.0149} C_DIS
LIN {X -56.6586,Y -5.5718,Z 68,A 178.6073,B 24.8775,C -2.5548,E1 24.8403,E2 265.2905} C_DIS
LIN {X -56.9022,Y -1.8735,Z 68,A 174.6746,B 24.8767,C -2.5632,E1 24.8398,E2 269.2267} C_DIS
LIN {X -56.8705,Y 2.6731,Z 68,A 170.8531,B 24.8741,C -2.5898,E1 24.84,E2 273.0077} C_DIS
LIN {X -56.5255,Y 6.8004,Z 68,A 166.5967,B 24.8729,C -2.6015,E1 24.8411,E2 277.2617} C_DIS
LIN {X -56.2298,Y 8.9227,Z 68,A 164.1488,B 24.8727,C -2.6036,E1 24.8421,E2 279.7192} C_DIS
LIN {X -55.7425,Y 11.5819,Z 68,A 160.9897,B 24.8726,C -2.605,E1 24.8438,E2 282.8935} C_DIS
LIN {X -55.0513,Y 14.5155,Z 68,A 157.8687,B 24.8718,C -2.613,E1 24.846,E2 286.0136} C_DIS
LIN {X -54.1221,Y 17.6684,Z 68,A 154.3621,B 24.8711,C -2.62,E1 24.8489,E2 289.5237} C_DIS
LIN {X -52.6603,Y 21.6397,Z 68,A 150.954,B 24.8685,C -2.6466,E1 24.8523,E2 292.8874} C_DIS
LIN {X -50.8993,Y 25.5083,Z 68,A 146.3896,B 24.8677,C -2.6544,E1 24.8577,E2 297.4579} C_DIS
LIN {X -49.5822,Y 27.9825,Z 68,A 143.5556,B 24.8669,C -2.6623,E1 24.8615,E2 300.2881} C_DIS
LIN {X -47.4124,Y 31.5192,Z 68,A 139.0839,B 24.8662,C -2.669,E1 24.8682,E2 304.7664} C_DIS
LIN {X -45.6693,Y 33.996,Z 68,A 135.676,B 24.866,C -2.6711,E1 24.8738,E2 308.1857} C_DIS
LIN {X -43.165,Y 37.1241,Z 68,A 132.0582,B 24.8643,C -2.6883,E1 24.8803,E2 311.7792} C_DIS
LIN {X -41.0199,Y 39.4806,Z 68,A 128.9769,B 24.8633,C -2.6982,E1 24.8861,E2 314.8503} C_DIS
LIN {X -39.2633,Y 41.2288,Z 68,A 126.5839,B 24.8625,C -2.7057,E1 24.8909,E2 317.2353} C_DIS
LIN {X -37.3503,Y 42.9689,Z 68,A 123.7477,B 24.8623,C -2.7076,E1 24.8968,E2 320.0783} C_DIS
LIN {X -34.7588,Y 45.0907,Z 68,A 120.7581,B 24.8609,C -2.7212,E1 24.9033,E2 323.0465} C_DIS
LIN {X -33.3528,Y 46.1414,Z 68,A 118.3077,B 24.8618,C -2.713,E1 24.9089,E2 325.525} C_DIS
LIN {X -30.4362,Y 48.1152,Z 68,A 114.9332,B 24.8608,C -2.7226,E1 24.9168,E2 328.8877} C_DIS
LIN {X -27.2418,Y 49.9925,Z 68,A 111.9755,B 24.8587,C -2.7426,E1 24.9238,E2 331.8063} C_DIS
LIN {X -25.5883,Y 50.8596,Z 68,A 109.4319,B 24.8596,C -2.7339,E1 24.9302,E2 334.3777} C_DIS
LIN {X -23.4579,Y 51.8756,Z 68,A 106.8475,B 24.8596,C -2.7337,E1 24.9368,E2 336.9688} C_DIS
LIN {X -19.4635,Y 53.5026,Z 68,A 103.2705,B 24.8576,C -2.7533,E1 24.946,E2 340.5071} C_DIS
LIN {X -16.8253,Y 54.3899,Z 68,A 99.7905,B 24.8586,C -2.7442,E1 24.9553,E2 344.015} C_DIS
LIN {X -14.3083,Y 55.1057,Z 68,A 97.5854,B 24.8575,C -2.7547,E1 24.9612,E2 346.1986} C_DIS
LIN {X -10.9662,Y 55.8671,Z 68,A 94.0384,B 24.8574,C -2.7558,E1 24.9708,E2 349.7472} C_DIS
LIN {X -8.5919,Y 56.2809,Z 68,A 91.5426,B 24.8574,C -2.7562,E1 24.9777,E2 352.2444} C_DIS
LIN {X -6.1329,Y 56.602,Z 68,A 88.3608,B 24.8585,C -2.7448,E1 24.9866,E2 355.4554} C_DIS
LIN {X -0.3678,Y 56.9317,Z 68,A 83.4186,B 24.8566,C -2.7632,E1 25.0003,E2 360.355} C_DIS
LIN {X 1.716,Y 56.907,Z 68,A 81.2611,B 24.8566,C -2.7623,E1 25.0063,E2 362.5143} C_DIS
LIN {X 4.1436,Y 56.7827,Z 68,A 78.5939,B 24.8571,C -2.758,E1 25.0138,E2 365.1906} C_DIS
LIN {X 7.9383,Y 56.3768,Z 68,A 74.3026,B 24.8581,C -2.7486,E1 25.0257,E2 369.501} C_DIS
LIN {X 11.4946,Y 55.7604,Z 68,A 71.1045,B 24.8574,C -2.7556,E1 25.0344,E2 372.6787} C_DIS
LIN {X 14.0986,Y 55.1596,Z 68,A 67.7037,B 24.859,C -2.74,E1 25.0437,E2 376.1115} C_DIS
LIN {X 17.8244,Y 54.0716,Z 68,A 64.3514,B 24.8582,C -2.7481,E1 25.0526,E2 379.4385} C_DIS
LIN {X 20.9358,Y 52.9439,Z 68,A 61.1468,B 24.8582,C -2.7475,E1 25.061,E2 382.6375} C_DIS
LIN {X 23.3732,Y 51.9138,Z 68,A 58.5875,B 24.8582,C -2.7468,E1 25.0675,E2 385.1923} C_DIS
LIN {X 25.6466,Y 50.8298,Z 68,A 55.5613,B 24.8597,C -2.7336,E1 25.0751,E2 388.2418} C_DIS
LIN {X 29.2622,Y 48.8384,Z 68,A 51.6565,B 24.8597,C -2.7329,E1 25.0845,E2 392.1364} C_DIS
LIN {X 32.1356,Y 46.9965,Z 68,A 48.2024,B 24.8603,C -2.7271,E1 25.0926,E2 395.5928} C_DIS
LIN {X 34.1216,Y 45.575,Z 68,A 45.6802,B 24.8609,C -2.7215,E1 25.0983,E2 398.1192} C_DIS
LIN {X 36.9621,Y 43.3031,Z 68,A 41.9415,B 24.8618,C -2.7131,E1 25.1063,E2 401.8636} C_DIS
LIN {X 39.5996,Y 40.9052,Z 68,A 38.795,B 24.8615,C -2.7153,E1 25.1127,E2 404.992} C_DIS
LIN {X 42.191,Y 38.2281,Z 68,A 35.0377,B 24.8624,C -2.707,E1 25.1199,E2 408.7525} C_DIS
LIN {X 44.1333,Y 35.967,Z 68,A 32.2073,B 24.8627,C -2.7039,E1 25.1249,E2 411.5773} C_DIS
LIN {X 46.4039,Y 32.9854,Z 68,A 28.0617,B 24.8645,C -2.6866,E1 25.1319,E2 415.7439} C_DIS
LIN {X 47.9492,Y 30.6958,Z 68,A 25.7941,B 24.864,C -2.6909,E1 25.1353,E2 417.9901} C_DIS
LIN {X 49.1909,Y 28.6658,Z 68,A 23.1831,B 24.8651,C -2.6799,E1 25.1391,E2 420.6138} C_DIS
LIN {X 50.597,Y 26.1025,Z 68,A 20.2732,B 24.8659,C -2.6727,E1 25.1429,E2 423.5254} C_DIS
LIN {X 51.8445,Y 23.5271,Z 68,A 17.8407,B 24.8657,C -2.6747,E1 25.1458,E2 425.9399} C_DIS
LIN {X 52.9746,Y 20.8576,Z 68,A 14.1208,B 24.8683,C -2.6485,E1 25.1498,E2 429.7013} C_DIS
LIN {X 53.8409,Y 18.51,Z 68,A 11.2396,B 24.8698,C -2.6331,E1 25.1524,E2 432.6028} C_DIS
LIN {X 54.8363,Y 15.3095,Z 68,A 8.6429,B 24.8691,C -2.6404,E1 25.1544,E2 435.1674} C_DIS
LIN {X 55.5325,Y 12.5526,Z 68,A 5.7599,B 24.87,C -2.6313,E1 25.1563,E2 438.0552} C_DIS
LIN {X 56.1954,Y 9.1373,Z 68,A 2.0636,B 24.8715,C -2.6162,E1 25.1581,E2 441.7656} C_DIS
LIN {X 56.5917,Y 6.2305,Z 68,A -0.6408,B 24.8718,C -2.6126,E1 25.159,E2 444.4625} C_DIS
LIN {X 56.8811,Y 2.427,Z 68,A -4.5952,B 24.8733,C -2.598,E1 25.1597,E2 448.428} C_DIS
LIN {X 56.9345,Y -0.1802,Z 68,A -6.9248,B 24.8734,C -2.5964,E1 25.1597,E2 450.7476} C_DIS
LIN {X 56.8767,Y -2.5302,Z 68,A -9.7588,B 24.8752,C -2.5783,E1 25.1595,E2 453.6074} C_DIS
LIN {X 56.6603,Y -5.5746,Z 68,A -12.2124,B 24.8748,C -2.5826,E1 25.1589,E2 456.0363} C_DIS
LIN {X 56.2235,Y -8.9631,Z 68,A -15.5172,B 24.8755,C -2.5748,E1 25.1577,E2 459.3401} C_DIS
LIN {X 55.7677,Y -11.4592,Z 68,A -18.7843,B 24.8779,C -2.5506,E1 25.1559,E2 462.6452} C_DIS
LIN {X 55.0244,Y -14.6191,Z 68,A -21.6458,B 24.8779,C -2.5496,E1 25.1539,E2 465.4926} C_DIS
LIN {X 54.2553,Y -17.2567,Z 68,A -24.342,B 24.8786,C -2.5426,E1 25.1517,E2 468.1899} C_DIS
LIN {X 53.363,Y -19.8457,Z 68,A -27.2008,B 24.8797,C -2.5319,E1 25.149,E2 471.058} C_DIS
LIN {X 51.7977,Y -23.6309,Z 68,A -30.9756,B 24.8801,C -2.5275,E1 25.1449,E2 474.8227} C_DIS
LIN {X 51.0365,Y -25.2315,Z 68,A -33.1125,B 24.8813,C -2.5143,E1 25.1423,E2 476.9794} C_DIS
LIN {X 49.3472,Y -28.3937,Z 68,A -36.2557,B 24.8813,C -2.5143,E1 25.1381,E2 480.1058} C_DIS
LIN {X 47.8978,Y -30.7758,Z 68,A -39.7734,B 24.8836,C -2.4906,E1 25.1328,E2 483.6619} C_DIS
LIN {X 46.202,Y -33.2681,Z 68,A -42.8675,B 24.8845,C -2.481,E1 25.1278,E2 486.7635} C_DIS
LIN {X 43.452,Y -36.7873,Z 68,A -46.9744,B 24.8847,C -2.478,E1 25.1206,E2 490.8586} C_DIS
LIN {X 40.8468,Y -39.6602,Z 68,A -50.2957,B 24.8844,C -2.4812,E1 25.1143,E2 494.1576} C_DIS
LIN {X 39.4934,Y -41.0076,Z 68,A -52.6869,B 24.8858,C -2.4663,E1 25.1095,E2 496.5741} C_DIS
LIN {X 37.1001,Y -43.1853,Z 68,A -55.7238,B 24.8861,C -2.4638,E1 25.1032,E2 499.605} C_DIS
LIN {X 34.7315,Y -45.1118,Z 68,A -59.2505,B 24.8876,C -2.4473,E1 25.0954,E2 503.1575} C_DIS
LIN {X 32.2802,Y -46.8979,Z 68,A -62.4503,B 24.8884,C -2.4381,E1 25.0881,E2 506.3682} C_DIS
LIN {X 28.4689,Y -49.304,Z 68,A -66.1855,B 24.8876,C -2.4469,E1 25.0793,E2 510.0707} C_DIS
LIN {X 26.1472,Y -50.5741,Z 68,A -69.3198,B 24.889,C -2.4324,E1 25.0715,E2 513.2306} C_DIS
LIN {X 23.7989,Y -51.7206,Z 68,A -71.5234,B 24.8885,C -2.4373,E1 25.0659,E2 515.4167} C_DIS
LIN {X 20.5831,Y -53.0825,Z 68,A -74.9522,B 24.8888,C -2.4341,E1 25.0571,E2 518.8451} C_DIS
LIN {X 16.6189,Y -54.4539,Z 68,A -79.0847,B 24.8891,C -2.4308,E1 25.0462,E2 522.9774} C_DIS
LIN {X 14.8082,Y -54.9734,Z 68,A -81.3636,B 24.89,C -2.4208,E1 25.04,E2 525.2763} C_DIS
LIN {X 12.0839,Y -55.6357,Z 68,A -84.4764,B 24.8908,C -2.4122,E1 25.0315,E2 528.4052} C_DIS
LIN {X 8.1689,Y -56.344,Z 68,A -87.6621,B 24.8896,C -2.4259,E1 25.0228,E2 531.555} C_DIS
LIN {X 6.3296,Y -56.5807,Z 68,A -90.3914,B 24.8912,C -2.4073,E1 25.0151,E2 534.3265} C_DIS
LIN {X 3.011,Y -56.8533,Z 68,A -93.3261,B 24.8906,C -2.4142,E1 25.007,E2 537.2437} C_DIS
LIN {X 0.3066,Y -56.9308,Z 68,A -94.7875,B 24.8884,C -2.4387,E1 25.0031,E2 538.6464} C_DIS
Enddeposition()
LIN {X 0.3066,Y -56.9308,Z 68,A -94.7875,B 24.8884,C -2.4387,E1 25.0031,E2 538.6464} C_DIS
Startdeposition()
$VEL.CP = VEL_PRINT
LIN {X 1.5091,Y -55.969,Z 68,A -93.6531,B 24.887,C -2.4533,E1 25.0064,E2 537.4776} C_DIS
LIN {X 3.7737,Y -55.8618,Z 68,A -90.5921,B 24.8856,C -2.4693,E1 25.015,E2 534.3799} C_DIS
LIN {X 7.949,Y -55.422,Z 68,A -86.049,B 24.8848,C -2.4771,E1 25.0276,E2 529.8219} C_DIS
LIN {X 11.1454,Y -54.8687,Z 68,A -83.8211,B 24.8867,C -2.4573,E1 25.0336,E2 527.6438} C_DIS
LIN {X 14.8403,Y -53.9871,Z 68,A -79.7754,B 24.886,C -2.4644,E1 25.0446,E2 523.5873} C_DIS
LIN {X 17.9379,Y -53.0379,Z 68,A -76.4837,B 24.8857,C -2.4678,E1 25.0533,E2 520.2936} C_DIS
LIN {X 20.3955,Y -52.1422,Z 68,A -74.003,B 24.8857,C -2.4672,E1 25.0598,E2 517.8196} C_DIS
LIN {X 22.2107,Y -51.3955,Z 68,A -71.8807,B 24.8853,C -2.4725,E1 25.0652,E2 515.6898} C_DIS
LIN {X 24.3963,Y -50.3947,Z 68,A -69.3065,B 24.8847,C -2.4788,E1 25.0718,E2 513.1074} C_DIS
LIN {X 27.0813,Y -49.0044,Z 68,A -66.261,B 24.8843,C -2.4829,E1 25.0793,E2 510.0607} C_DIS
LIN {X 29.5157,Y -47.5777,Z 68,A -63.2949,B 24.8836,C -2.4899,E1 25.0864,E2 507.0872} C_DIS
LIN {X 31.5353,Y -46.2637,Z 68,A -61.2608,B 24.8841,C -2.4853,E1 25.0911,E2 505.0708} C_DIS
LIN {X 33.8637,Y -44.5883,Z 68,A -57.5711,B 24.8819,C -2.5078,E1 25.0994,E2 501.341} C_DIS
LIN {X 37.592,Y -41.4938,Z 68,A -52.5745,B 24.8808,C -2.5197,E1 25.11,E2 496.3358} C_DIS
LIN {X 41.0448,Y -38.0814,Z 68,A -47.5093,B 24.8795,C -2.5339,E1 25.1198,E2 491.2588} C_DIS
LIN {X 44.1835,Y -34.3899,Z 68,A -42.7845,B 24.8787,C -2.5415,E1 25.1282,E2 486.538} C_DIS
LIN {X 45.8895,Y -32.0774,Z 68,A -40.4932,B 24.8794,C -2.5348,E1 25.1318,E2 484.2736} C_DIS
LIN {X 47.2201,Y -30.0845,Z 68,A -37.8138,B 24.8782,C -2.5467,E1 25.136,E2 481.5796} C_DIS
LIN {X 48.6672,Y -27.6827,Z 68,A -34.9071,B 24.8774,C -2.5557,E1 25.1401,E2 478.6665} C_DIS
LIN {X 50.0757,Y -25.0448,Z 68,A -32.0607,B 24.877,C -2.5597,E1 25.1437,E2 475.8257} C_DIS
LIN {X 51.0984,Y -22.8855,Z 68,A -29.7344,B 24.8766,C -2.5642,E1 25.1464,E2 473.5012} C_DIS
LIN {X 51.8608,Y -21.1006,Z 68,A -26.8786,B 24.8741,C -2.59,E1 25.1495,E2 470.6002} C_DIS
LIN {X 53.2875,Y -17.182,Z 68,A -23.2871,B 24.8743,C -2.5876,E1 25.1527,E2 467.0347} C_DIS
LIN {X 54.3756,Y -13.3447,Z 68,A -19.5101,B 24.8737,C -2.5933,E1 25.1555,E2 463.266} C_DIS
LIN {X 54.7468,Y -11.7296,Z 68,A -17.0729,B 24.8716,C -2.6155,E1 25.1569,E2 460.7903} C_DIS
LIN {X 55.2725,Y -8.9344,Z 68,A -13.5735,B 24.8693,C -2.6383,E1 25.1585,E2 457.2577} C_DIS
LIN {X 55.7341,Y -5.3413,Z 68,A -11.2528,B 24.8713,C -2.6181,E1 25.1592,E2 454.9984} C_DIS
LIN {X 55.8785,Y -3.5149,Z 68,A -9.2385,B 24.8704,C -2.6272,E1 25.1596,E2 452.9746} C_DIS
LIN {X 55.974,Y -1.3283,Z 68,A -6.9817,B 24.8697,C -2.6347,E1 25.1598,E2 450.7136} C_DIS
LIN {X 55.9715,Y 1.4007,Z 68,A -4.1551,B 24.8687,C -2.6442,E1 25.1597,E2 447.8811} C_DIS
LIN {X 55.8212,Y 4.3343,Z 68,A -1.2848,B 24.8681,C -2.6506,E1 25.1592,E2 445.013} C_DIS
LIN {X 55.5556,Y 6.9581,Z 68,A 1.8197,B 24.8663,C -2.6682,E1 25.1582,E2 441.8852} C_DIS
LIN {X 54.7863,Y 11.5469,Z 68,A 5.9244,B 24.8663,C -2.6678,E1 25.1562,E2 437.8053} C_DIS
LIN {X 54.3441,Y 13.4737,Z 68,A 8.2494,B 24.865,C -2.6808,E1 25.1546,E2 435.4632} C_DIS
LIN {X 53.4491,Y 16.6728,Z 68,A 11.9514,B 24.8633,C -2.6977,E1 25.1517,E2 431.7423} C_DIS
LIN {X 52.7119,Y 18.8772,Z 68,A 14.2723,B 24.8628,C -2.7033,E1 25.1495,E2 429.4213} C_DIS
LIN {X 51.3461,Y 22.324,Z 68,A 17.5136,B 24.8629,C -2.7016,E1 25.1461,E2 426.2016} C_DIS
LIN {X 50.0098,Y 25.1764,Z 68,A 20.5854,B 24.8624,C -2.7071,E1 25.1424,E2 423.1334} C_DIS
LIN {X 49.0993,Y 26.9091,Z 68,A 22.7918,B 24.8614,C -2.717,E1 25.1395,E2 420.9152} C_DIS
LIN {X 48.0025,Y 28.8206,Z 68,A 25.4391,B 24.8599,C -2.7316,E1 25.1357,E2 418.247} C_DIS
LIN {X 46.4969,Y 31.1906,Z 68,A 28.3172,B 24.8591,C -2.7389,E1 25.1313,E2 415.3658} C_DIS
LIN {X 44.1713,Y 34.4059,Z 68,A 31.7923,B 24.8594,C -2.7358,E1 25.1255,E2 411.9147} C_DIS
LIN {X 42.2014,Y 36.7943,Z 68,A 35.1756,B 24.8582,C -2.7477,E1 25.1194,E2 408.5188} C_DIS
LIN {X 39.3744,Y 39.805,Z 68,A 39.2675,B 24.8576,C -2.7538,E1 25.1115,E2 404.4301} C_DIS
LIN {X 36.1967,Y 42.7153,Z 68,A 43.5478,B 24.857,C -2.7597,E1 25.1027,E2 400.1532} C_DIS
LIN {X 33.664,Y 44.7383,Z 68,A 47.2128,B 24.8556,C -2.773,E1 25.0946,E2 396.4701} C_DIS
LIN {X 31.2944,Y 46.4269,Z 68,A 50.1156,B 24.8552,C -2.7763,E1 25.0879,E2 393.5696} C_DIS
LIN {X 28.4508,Y 48.2217,Z 68,A 53.5882,B 24.8546,C -2.782,E1 25.0796,E2 390.0942} C_DIS
LIN {X 25.427,Y 49.8824,Z 68,A 57.3898,B 24.8535,C -2.7922,E1 25.0702,E2 386.2791} C_DIS
LIN {X 22.2459,Y 51.3802,Z 68,A 60.5743,B 24.854,C -2.7877,E1 25.0622,E2 383.1132} C_DIS
LIN {X 20.2007,Y 52.2187,Z 68,A 62.9524,B 24.8535,C -2.7923,E1 25.056,E2 380.7297} C_DIS
LIN {X 17.4336,Y 53.2061,Z 68,A 65.6441,B 24.8539,C -2.7885,E1 25.0489,E2 378.0524} C_DIS
LIN {X 15.5711,Y 53.7807,Z 68,A 68.5559,B 24.8518,C -2.8084,E1 25.041,E2 375.0983} C_DIS
LIN {X 12.282,Y 54.6264,Z 68,A 71.4565,B 24.8529,C -2.7987,E1 25.0332,E2 372.2248} C_DIS
LIN {X 8.8495,Y 55.2857,Z 68,A 75.0122,B 24.8528,C -2.7995,E1 25.0234,E2 368.6709} C_DIS
LIN {X 5.8934,Y 55.6781,Z 68,A 78.123,B 24.8526,C -2.8013,E1 25.0148,E2 365.5583} C_DIS
LIN {X 3.1679,Y 55.8995,Z 68,A 80.8467,B 24.8527,C -2.7998,E1 25.0072,E2 362.8393} C_DIS
LIN {X 0.6513,Y 55.9862,Z 68,A 83.8742,B 24.8519,C -2.8082,E1 24.9987,E2 359.7923} C_DIS
LIN {X -3.5774,Y 55.8751,Z 68,A 88.3025,B 24.8519,C -2.8086,E1 24.9864,E2 355.3619} C_DIS
LIN {X -7.1619,Y 55.5292,Z 68,A 91.068,B 24.8539,C -2.7892,E1 24.9788,E2 352.6408} C_DIS
LIN {X -9.1988,Y 55.2283,Z 68,A 93.4795,B 24.8534,C -2.7935,E1 24.9721,E2 350.2171} C_DIS
LIN {X -12.468,Y 54.5834,Z 68,A 97.1033,B 24.8533,C -2.7946,E1 24.9622,E2 346.5863} C_DIS
LIN {X -14.8573,Y 53.9825,Z 68,A 99.7401,B 24.8533,C -2.7942,E1 24.9551,E2 343.9464} C_DIS
LIN {X -18.2318,Y 52.9381,Z 68,A 102.8063,B 24.8548,C -2.78,E1 24.947,E2 340.9085} C_DIS
LIN {X -21.1467,Y 51.8421,Z 68,A 106.1326,B 24.855,C -2.7783,E1 24.9383,E2 337.5791} C_DIS
LIN {X -23.116,Y 50.9946,Z 68,A 109.212,B 24.8537,C -2.791,E1 24.9304,E2 334.462} C_DIS
LIN {X -26.8641,Y 49.1237,Z 68,A 113.1249,B 24.8551,C -2.7773,E1 24.9208,E2 330.571} C_DIS
LIN {X -30.1344,Y 47.1881,Z 68,A 116.4183,B 24.8569,C -2.7598,E1 24.913,E2 327.3091} C_DIS
LIN {X -32.6557,Y 45.4798,Z 68,A 119.7707,B 24.8571,C -2.7578,E1 24.9053,E2 323.9501} C_DIS
LIN {X -34.5648,Y 44.0459,Z 68,A 122.2671,B 24.8576,C -2.7537,E1 24.8998,E2 321.4545} C_DIS
LIN {X -36.6697,Y 42.3103,Z 68,A 124.9286,B 24.8584,C -2.7453,E1 24.8941,E2 318.8026} C_DIS
LIN {X -38.2239,Y 40.9115,Z 68,A 127.0276,B 24.859,C -2.7398,E1 24.8898,E2 316.7084} C_DIS
LIN {X -40.3609,Y 38.8045,Z 68,A 130.7247,B 24.8587,C -2.7431,E1 24.8825,E2 312.9876} C_DIS
LIN {X -42.5402,Y 36.4023,Z 68,A 134.7388,B 24.8583,C -2.7466,E1 24.8752,E2 308.9468} C_DIS
LIN {X -44.7438,Y 33.6568,Z 68,A 136.9985,B 24.8616,C -2.7146,E1 24.8714,E2 306.753} C_DIS
LIN {X -46.7339,Y 30.8339,Z 68,A 140.6235,B 24.8624,C -2.7065,E1 24.8657,E2 303.1294} C_DIS
LIN {X -47.786,Y 29.177,Z 68,A 143.014,B 24.8624,C -2.7073,E1 24.8621,E2 300.7249} C_DIS
LIN {X -49.157,Y 26.8026,Z 68,A 145.7292,B 24.8633,C -2.6978,E1 24.8584,E2 298.0182} C_DIS
LIN {X -50.7619,Y 23.6223,Z 68,A 149.6553,B 24.8639,C -2.6918,E1 24.8536,E2 294.0852} C_DIS
LIN {X -51.7025,Y 21.4873,Z 68,A 152.2568,B 24.8643,C -2.6882,E1 24.8508,E2 291.4779} C_DIS
LIN {X -53.1883,Y 17.4886,Z 68,A 155.9178,B 24.8668,C -2.6634,E1 24.8474,E2 287.8554} C_DIS
LIN {X -53.6708,Y 15.9443,Z 68,A 157.8216,B 24.8669,C -2.6623,E1 24.8459,E2 285.9431} C_DIS
LIN {X -54.3679,Y 13.3761,Z 68,A 160.6443,B 24.8676,C -2.6555,E1 24.8439,E2 283.1202} C_DIS
LIN {X -55.019,Y 10.3795,Z 68,A 163.4525,B 24.8691,C -2.6403,E1 24.8424,E2 280.3317} C_DIS
LIN {X -55.3965,Y 8.1283,Z 68,A 166.7128,B 24.8683,C -2.6481,E1 24.841,E2 277.0335} C_DIS
LIN {X -55.9034,Y 3.0961,Z 68,A 171.9746,B 24.8698,C -2.6332,E1 24.8399,E2 271.7758} C_DIS
LIN {X -55.9443,Y -2.2455,Z 68,A 176.3052,B 24.8733,C -2.5974,E1 24.8399,E2 267.5045} C_DIS
LIN {X -55.8132,Y -4.4343,Z 68,A 179.1212,B 24.8731,C -2.5997,E1 24.8405,E2 264.6662} C_DIS
LIN {X -55.5171,Y -7.2549,Z 68,A -178.178,B 24.8743,C -2.5874,E1 24.8413,E2 261.9786} C_DIS
LIN {X -55.1996,Y -9.3702,Z 68,A -175.281,B 24.8738,C -2.5923,E1 24.8427,E2 259.0527} C_DIS
LIN {X -54.0285,Y -14.687,Z 68,A -169.61,B 24.8753,C -2.5772,E1 24.8464,E2 253.3847} C_DIS
LIN {X -53.1074,Y -17.7292,Z 68,A -167.1284,B 24.8775,C -2.5548,E1 24.8485,E2 250.9423} C_DIS
LIN {X -52.525,Y -19.3894,Z 68,A -164.5884,B 24.8768,C -2.5619,E1 24.851,E2 248.3709} C_DIS
LIN {X -51.1166,Y -22.8437,Z 68,A -161.0725,B 24.8783,C -2.5462,E1 24.8548,E2 244.8733} C_DIS
LIN {X -50.0146,Y -25.168,Z 68,A -158.5659,B 24.8792,C -2.5368,E1 24.8579,E2 242.3755} C_DIS
LIN {X -47.6404,Y -29.4153,Z 68,A -153.9729,B 24.8811,C -2.5172,E1 24.8643,E2 237.8053} C_DIS
LIN {X -45.4261,Y -32.731,Z 68,A -149.4858,B 24.8814,C -2.514,E1 24.8713,E2 233.3036} C_DIS
LIN {X -43.8909,Y -34.7616,Z 68,A -147.0315,B 24.8822,C -2.5053,E1 24.8755,E2 230.8585} C_DIS
LIN {X -42.2987,Y -36.6826,Z 68,A -144.1664,B 24.8822,C -2.5049,E1 24.8807,E2 227.9813} C_DIS
LIN {X -40.4739,Y -38.6872,Z 68,A -141.3579,B 24.8827,C -2.4995,E1 24.8861,E2 225.1732} C_DIS
LIN {X -38.2916,Y -40.8478,Z 68,A -138.4421,B 24.8837,C -2.4892,E1 24.8919,E2 222.27} C_DIS
LIN {X -36.4012,Y -42.5411,Z 68,A -135.9219,B 24.8843,C -2.4829,E1 24.8972,E2 219.755} C_DIS
LIN {X -33.5536,Y -44.821,Z 68,A -132.2396,B 24.885,C -2.4754,E1 24.9053,E2 216.077} C_DIS
LIN {X -31.9349,Y -45.9885,Z 68,A -129.9433,B 24.8849,C -2.4766,E1 24.9105,E2 213.7699} C_DIS
LIN {X -29.6599,Y -47.4876,Z 68,A -126.1851,B 24.8836,C -2.4902,E1 24.9195,E2 209.9674} C_DIS
LIN {X -26.7823,Y -49.1681,Z 68,A -124.2994,B 24.8866,C -2.4576,E1 24.9239,E2 208.1538} C_DIS
LIN {X -24.5533,Y -50.319,Z 68,A -121.3606,B 24.8863,C -2.4612,E1 24.9313,E2 205.1985} C_DIS
LIN {X -23.0181,Y -51.0387,Z 68,A -119.2474,B 24.8858,C -2.4663,E1 24.9367,E2 203.0679} C_DIS
LIN {X -19.7165,Y -52.4028,Z 68,A -115.8619,B 24.8866,C -2.4578,E1 24.9454,E2 199.6954} C_DIS
LIN {X -16.1153,Y -53.6201,Z 68,A -111.8989,B 24.8868,C -2.4562,E1 24.956,E2 195.729} C_DIS
LIN {X -13.4943,Y -54.3391,Z 68,A -108.2528,B 24.8854,C -2.4713,E1 24.9659,E2 192.0417} C_DIS
LIN {X -8.738,Y -55.3034,Z 68,A -104.3459,B 24.8874,C -2.4489,E1 24.9765,E2 188.1839} C_DIS
LIN {X -6.8162,Y -55.5735,Z 68,A -102.1387,B 24.8871,C -2.4529,E1 24.9827,E2 185.9656} C_DIS
LIN {X -3.7422,Y -55.8639,Z 68,A -99.0591,B 24.8872,C -2.4512,E1 24.9912,E2 182.8887} C_DIS
LIN {X -1.128,Y -55.9778,Z 68,A -96.189,B 24.8868,C -2.4554,E1 24.9993,E2 180.0082} C_DIS
LIN {X -1.128,Y -55.9778,Z 68,A -96.189,B 24.8868,C -2.4554,E1 24.9993,E2 180.0082} C_DIS
Enddeposition()
LIN {X 0.3193,Y -55.0407,Z 68,A -96.1921,B 24.888,C -2.4431,E1 24.9992,E2 180.0404} C_DIS
Startdeposition()
$VEL.CP = VEL_PRINT
LIN {X -3.4517,Y -54.9376,Z 68,A -100.399,B 24.8885,C -2.4374,E1 24.9874,E2 184.2619} C_DIS
LIN {X -6.772,Y -54.628,Z 68,A -104.0196,B 24.8887,C -2.435,E1 24.9773,E2 187.8904} C_DIS
LIN {X -10.0962,Y -54.112,Z 68,A -107.2644,B 24.8882,C -2.4409,E1 24.9684,E2 191.1244} C_DIS
LIN {X -13.9131,Y -53.2585,Z 68,A -111.0887,B 24.8876,C -2.4475,E1 24.9581,E2 194.9382} C_DIS
LIN {X -16.5007,Y -52.5134,Z 68,A -114.0841,B 24.8877,C -2.4459,E1 24.9501,E2 197.9424} C_DIS
LIN {X -19.5238,Y -51.4666,Z 68,A -117.3338,B 24.8873,C -2.4502,E1 24.9415,E2 201.1884} C_DIS
LIN {X -22.2971,Y -50.3274,Z 68,A -120.2659,B 24.8867,C -2.4568,E1 24.934,E2 204.1116} C_DIS
LIN {X -24.2434,Y -49.4196,Z 68,A -122.8266,B 24.887,C -2.4536,E1 24.9275,E2 206.6864} C_DIS
LIN {X -27.0729,Y -47.9281,Z 68,A -126.4996,B 24.8872,C -2.4521,E1 24.9185,E2 210.3737} C_DIS
LIN {X -29.983,Y -46.1638,Z 68,A -129.8929,B 24.8864,C -2.4599,E1 24.9105,E2 213.7591} C_DIS
LIN {X -32.1094,Y -44.7102,Z 68,A -133.2274,B 24.887,C -2.4533,E1 24.9029,E2 217.1209} C_DIS
LIN {X -34.7445,Y -42.6945,Z 68,A -135.9683,B 24.8854,C -2.4715,E1 24.897,E2 219.8288} C_DIS
LIN {X -36.9217,Y -40.8271,Z 68,A -138.5352,B 24.8842,C -2.4842,E1 24.8917,E2 222.3755} C_DIS
LIN {X -38.4412,Y -39.3996,Z 68,A -140.8463,B 24.884,C -2.4862,E1 24.887,E2 224.6913} C_DIS
LIN {X -40.1641,Y -37.6409,Z 68,A -143.4423,B 24.8835,C -2.4911,E1 24.882,E2 227.2869} C_DIS
LIN {X -42.5397,Y -34.9352,Z 68,A -147.4355,B 24.8831,C -2.4955,E1 24.8747,E2 231.2878} C_DIS
LIN {X -44.7456,Y -32.0598,Z 68,A -151.9047,B 24.8833,C -2.4934,E1 24.8673,E2 235.7837} C_DIS
LIN {X -46.7786,Y -29.0136,Z 68,A -155.2824,B 24.8817,C -2.51,E1 24.8623,E2 239.1389} C_DIS
LIN {X -48.7883,Y -25.4897,Z 68,A -158.7556,B 24.8795,C -2.5332,E1 24.8577,E2 242.5749} C_DIS
LIN {X -50.0061,Y -23.0076,Z 68,A -162.2249,B 24.8797,C -2.5316,E1 24.8535,E2 246.0667} C_DIS
LIN {X -51.1705,Y -20.2856,Z 68,A -165.3362,B 24.8789,C -2.5399,E1 24.8502,E2 249.1756} C_DIS
LIN {X -52.38,Y -16.9212,Z 68,A -169.2283,B 24.8781,C -2.5481,E1 24.8467,E2 253.0703} C_DIS
LIN {X -53.5179,Y -12.8757,Z 68,A -173.2376,B 24.8763,C -2.5668,E1 24.8438,E2 257.0581} C_DIS
LIN {X -53.9744,Y -10.8084,Z 68,A -175.7336,B 24.8761,C -2.569,E1 24.8424,E2 259.5637} C_DIS
LIN {X -54.5308,Y -7.5122,Z 68,A -179.11,B 24.8749,C -2.5813,E1 24.841,E2 262.9308} C_DIS
LIN {X -54.8866,Y -4.1688,Z 68,A 177.3995,B 24.8738,C -2.5924,E1 24.8401,E2 266.4158} C_DIS
LIN {X -55.0167,Y -1.7787,Z 68,A 174.5073,B 24.8737,C -2.594,E1 24.8398,E2 269.3215} C_DIS
LIN {X -54.9542,Y 3.1686,Z 68,A 169.4122,B 24.872,C -2.6111,E1 24.8402,E2 274.4064} C_DIS
LIN {X -54.5747,Y 7.1825,Z 68,A 165.5046,B 24.8702,C -2.6288,E1 24.8414,E2 278.2952} C_DIS
LIN {X -54.2992,Y 9.0326,Z 68,A 163.1191,B 24.8703,C -2.6281,E1 24.8425,E2 280.6963} C_DIS
LIN {X -53.4401,Y 13.1974,Z 68,A 159.3492,B 24.8679,C -2.652,E1 24.8448,E2 284.4312} C_DIS
LIN {X -52.9234,Y 15.1369,Z 68,A 157.1232,B 24.8675,C -2.6564,E1 24.8465,E2 286.6598} C_DIS
LIN {X -52.2539,Y 17.3087,Z 68,A 154.4782,B 24.8672,C -2.6593,E1 24.8487,E2 289.3131} C_DIS
LIN {X -51.0355,Y 20.6248,Z 68,A 151.2571,B 24.8654,C -2.6774,E1 24.8519,E2 292.5088} C_DIS
LIN {X -49.6906,Y 23.6826,Z 68,A 147.1262,B 24.8654,C -2.6774,E1 24.8567,E2 296.6622} C_DIS
LIN {X -48.4034,Y 26.2127,Z 68,A 144.2847,B 24.8643,C -2.6877,E1 24.8604,E2 299.4943} C_DIS
LIN {X -46.7732,Y 29.0221,Z 68,A 141.0879,B 24.8631,C -2.7001,E1 24.865,E2 302.678} C_DIS
LIN {X -45.1973,Y 31.4196,Z 68,A 137.875,B 24.8626,C -2.7046,E1 24.87,E2 305.8959} C_DIS
LIN {X -43.8182,Y 33.3176,Z 68,A 135.3967,B 24.862,C -2.7105,E1 24.8742,E2 308.3722} C_DIS
LIN {X -41.6233,Y 36.0209,Z 68,A 132.369,B 24.8601,C -2.7293,E1 24.8795,E2 311.3689} C_DIS
LIN {X -39.6549,Y 38.177,Z 68,A 128.3342,B 24.861,C -2.7207,E1 24.8873,E2 315.4421} C_DIS
LIN {X -35.9891,Y 41.6517,Z 68,A 123.7289,B 24.8587,C -2.7432,E1 24.8967,E2 320.0122} C_DIS
LIN {X -34.37,Y 42.9971,Z 68,A 121.3471,B 24.8585,C -2.7447,E1 24.9019,E2 322.3993} C_DIS
LIN {X -31.9583,Y 44.818,Z 68,A 118.5453,B 24.8573,C -2.7568,E1 24.9081,E2 325.1822} C_DIS
LIN {X -30.5846,Y 45.7671,Z 68,A 116.6095,B 24.8573,C -2.7568,E1 24.9126,E2 327.1244} C_DIS
LIN {X -28.7065,Y 46.9673,Z 68,A 113.6356,B 24.8579,C -2.7502,E1 24.9197,E2 330.1234} C_DIS
LIN {X -25.9668,Y 48.5367,Z 68,A 109.9049,B 24.8581,C -2.7482,E1 24.9289,E2 333.8693} C_DIS
LIN {X -23.0061,Y 50.0077,Z 68,A 107.8879,B 24.8551,C -2.7776,E1 24.9339,E2 335.8215} C_DIS
LIN {X -20.6124,Y 51.0405,Z 68,A 104.4021,B 24.8561,C -2.7681,E1 24.9429,E2 339.3378} C_DIS
LIN {X -17.4276,Y 52.2136,Z 68,A 101.1622,B 24.8551,C -2.7775,E1 24.9514,E2 342.5616} C_DIS
LIN {X -14.6329,Y 53.0655,Z 68,A 98.5094,B 24.854,C -2.7876,E1 24.9584,E2 345.1949} C_DIS
LIN {X -12.4072,Y 53.6288,Z 68,A 95.312,B 24.8553,C -2.7756,E1 24.9672,E2 348.4253} C_DIS
LIN {X -8.8958,Y 54.3221,Z 68,A 92.3468,B 24.8536,C -2.7919,E1 24.9753,E2 351.3546} C_DIS
LIN {X -6.7212,Y 54.6338,Z 68,A 89.7039,B 24.8541,C -2.7869,E1 24.9826,E2 354.0115} C_DIS
LIN {X -3.8091,Y 54.9135,Z 68,A 86.1096,B 24.855,C -2.7783,E1 24.9927,E2 357.6277} C_DIS
LIN {X 1.4289,Y 55.0274,Z 68,A 81.18,B 24.8539,C -2.7891,E1 25.0064,E2 362.5317} C_DIS
LIN {X 6.1348,Y 54.7031,Z 68,A 76.5528,B 24.8534,C -2.7941,E1 25.0192,E2 367.1446} C_DIS
LIN {X 8.7976,Y 54.3385,Z 68,A 73.0662,B 24.8548,C -2.7803,E1 25.0289,E2 370.6607} C_DIS
LIN {X 11.8513,Y 53.7546,Z 68,A 70.284,B 24.854,C -2.7875,E1 25.0365,E2 373.4223} C_DIS
LIN {X 14.8774,Y 52.9969,Z 68,A 66.8392,B 24.8547,C -2.7817,E1 25.0458,E2 376.8755} C_DIS
LIN {X 17.4773,Y 52.1971,Z 68,A 64.2828,B 24.8543,C -2.7848,E1 25.0525,E2 379.4197} C_DIS
LIN {X 19.462,Y 51.49,Z 68,A 61.9332,B 24.8549,C -2.7798,E1 25.0587,E2 381.7764} C_DIS
LIN {X 22.1077,Y 50.4108,Z 68,A 59.2503,B 24.8546,C -2.7824,E1 25.0656,E2 384.4467} C_DIS
LIN {X 23.9212,Y 49.5754,Z 68,A 56.9417,B 24.8553,C -2.7754,E1 25.0715,E2 386.7659} C_DIS
LIN {X 26.7205,Y 48.1251,Z 68,A 53.9616,B 24.8551,C -2.7772,E1 25.0788,E2 389.7334} C_DIS
LIN {X 29.5917,Y 46.415,Z 68,A 50.3671,B 24.8559,C -2.7698,E1 25.0874,E2 393.3343} C_DIS
LIN {X 32.3982,Y 44.5013,Z 68,A 46.7191,B 24.8567,C -2.7617,E1 25.0957,E2 396.9889} C_DIS
LIN {X 34.5626,Y 42.842,Z 68,A 43.9492,B 24.8571,C -2.758,E1 25.1018,E2 399.7572} C_DIS
LIN {X 36.6966,Y 41.0286,Z 68,A 40.6267,B 24.8586,C -2.744,E1 25.1088,E2 403.0997} C_DIS
LIN {X 39.6238,Y 38.2092,Z 68,A 36.6629,B 24.8589,C -2.7408,E1 25.1167,E2 407.0546} C_DIS
LIN {X 41.518,Y 36.1421,Z 68,A 33.7953,B 24.8595,C -2.7354,E1 25.122,E2 409.9222} C_DIS
LIN {X 43.0397,Y 34.3167,Z 68,A 30.9457,B 24.8609,C -2.7217,E1 25.127,E2 412.7908} C_DIS
LIN {X 44.9593,Y 31.7604,Z 68,A 28.2646,B 24.8603,C -2.7273,E1 25.1314,E2 415.4457} C_DIS
LIN {X 47.1962,Y 28.3302,Z 68,A 23.7985,B 24.8619,C -2.7121,E1 25.1381,E2 419.9253} C_DIS
LIN {X 48.8091,Y 25.4502,Z 68,A 20.7643,B 24.8619,C -2.7116,E1 25.1422,E2 422.9449} C_DIS
LIN {X 50.1804,Y 22.6257,Z 68,A 17.315,B 24.8632,C -2.6987,E1 25.1463,E2 426.4062} C_DIS
LIN {X 51.2515,Y 20.0816,Z 68,A 14.1246,B 24.8648,C -2.6836,E1 25.1497,E2 429.6145} C_DIS
LIN {X 52.0361,Y 17.953,Z 68,A 11.9841,B 24.865,C -2.6815,E1 25.1517,E2 431.748} C_DIS
LIN {X 53.2521,Y 13.9379,Z 68,A 7.5934,B 24.8663,C -2.6681,E1 25.1551,E2 436.1455} C_DIS
LIN {X 53.7227,Y 11.9972,Z 68,A 5.3456,B 24.8673,C -2.6581,E1 25.1565,E2 438.4037} C_DIS
LIN {X 54.3529,Y 8.7087,Z 68,A 2.1146,B 24.8678,C -2.653,E1 25.1581,E2 441.6279} C_DIS
LIN {X 54.7846,Y 5.3601,Z 68,A -1.326,B 24.8688,C -2.6437,E1 25.1592,E2 445.0703} C_DIS
LIN {X 54.9604,Y 3.0574,Z 68,A -3.5439,B 24.8691,C -2.6402,E1 25.1596,E2 447.283} C_DIS
LIN {X 55.046,Y 0.2825,Z 68,A -6.8958,B 24.871,C -2.621,E1 25.1598,E2 450.6606} C_DIS
LIN {X 54.9764,Y -2.7458,Z 68,A -9.9575,B 24.8718,C -2.613,E1 25.1594,E2 453.7228} C_DIS
LIN {X 54.6621,Y -6.4846,Z 68,A -14.0728,B 24.8735,C -2.5961,E1 25.1583,E2 457.8538} C_DIS
LIN {X 54.2927,Y -9.0715,Z 68,A -17.1524,B 24.8751,C -2.5797,E1 25.1569,E2 460.9541} C_DIS
LIN {X 53.4807,Y -13.031,Z 68,A -20.7376,B 24.8751,C -2.5801,E1 25.1546,E2 464.5174} C_DIS
LIN {X 52.3929,Y -16.8812,Z 68,A -24.0581,B 24.8745,C -2.5859,E1 25.1521,E2 467.8054} C_DIS
LIN {X 51.6202,Y -19.1153,Z 68,A -27.3958,B 24.8771,C -2.5591,E1 25.1489,E2 471.1877} C_DIS
LIN {X 50.3975,Y -22.1382,Z 68,A -30.5599,B 24.8775,C -2.554,E1 25.1455,E2 474.3466} C_DIS
LIN {X 49.1134,Y -24.8579,Z 68,A -33.4806,B 24.878,C -2.5494,E1 25.1419,E2 477.2624} C_DIS
LIN {X 47.9856,Y -26.9702,Z 68,A -35.8501,B 24.8784,C -2.5449,E1 25.1387,E2 479.6301} C_DIS
LIN {X 46.9854,Y -28.677,Z 68,A -38.1923,B 24.8796,C -2.5329,E1 25.1353,E2 481.9886} C_DIS
LIN {X 45.2184,Y -31.3893,Z 68,A -41.4292,B 24.8802,C -2.5266,E1 25.1303,E2 485.2245} C_DIS
LIN {X 43.3295,Y -33.95,Z 68,A -45.0156,B 24.8816,C -2.5119,E1 25.1242,E2 488.8286} C_DIS
LIN {X 41.5493,Y -36.1063,Z 68,A -47.8317,B 24.8821,C -2.5065,E1 25.1191,E2 491.6446} C_DIS
LIN {X 39.24,Y -38.6034,Z 68,A -50.8858,B 24.8819,C -2.5083,E1 25.1133,E2 494.6813} C_DIS
LIN {X 38.1389,Y -39.6916,Z 68,A -52.8988,B 24.8831,C -2.4959,E1 25.1092,E2 496.7151} C_DIS
LIN {X 35.6076,Y -41.9774,Z 68,A -56.014,B 24.883,C -2.4971,E1 25.1027,E2 499.8151} C_DIS
LIN {X 33.4231,Y -43.7371,Z 68,A -59.4839,B 24.8846,C -2.4793,E1 25.0951,E2 503.3143} C_DIS
LIN {X 30.8344,Y -45.5986,Z 68,A -62.6913,B 24.885,C -2.475,E1 25.0877,E2 506.5208} C_DIS
LIN {X 28.078,Y -47.3458,Z 68,A -65.6996,B 24.8849,C -2.4768,E1 25.0806,E2 509.5153} C_DIS
LIN {X 26.3536,Y -48.327,Z 68,A -67.8813,B 24.8854,C -2.4709,E1 25.0753,E2 511.7048} C_DIS
LIN {X 24.2054,Y -49.4382,Z 68,A -70.5114,B 24.886,C -2.4645,E1 25.0687,E2 514.343} C_DIS
LIN {X 21.4449,Y -50.6963,Z 68,A -73.5976,B 24.8863,C -2.4612,E1 25.0608,E2 517.4292} C_DIS
LIN {X 18.4195,Y -51.8725,Z 68,A -77.4822,B 24.8877,C -2.4466,E1 25.0505,E2 521.3403} C_DIS
LIN {X 15.7793,Y -52.7354,Z 68,A -80.2481,B 24.8877,C -2.4458,E1 25.0432,E2 524.1032} C_DIS
LIN {X 11.9896,Y -53.7244,Z 68,A -83.7356,B 24.887,C -2.4536,E1 25.0338,E2 527.5672} C_DIS
LIN {X 10.1958,Y -54.0926,Z 68,A -86.4577,B 24.8886,C -2.436,E1 25.0262,E2 530.3279} C_DIS
LIN {X 6.5329,Y -54.6565,Z 68,A -90.3905,B 24.889,C -2.4321,E1 25.0153,E2 534.2668} C_DIS
LIN {X 3.233,Y -54.9507,Z 68,A -93.1868,B 24.888,C -2.4431,E1 25.0076,E2 537.0357} C_DIS
LIN {X 0.6029,Y -55.0427,Z 68,A -96.1786,B 24.8885,C -2.4374,E1 24.9992,E2 540.0404} C_DIS
LIN {X 0.6029,Y -55.0427,Z 68,A -96.1786,B 24.8885,C -2.4374,E1 24.9992,E2 540.0404} C_DIS
Enddeposition()
LIN {X 0.3269,Y -54.0921,Z 68,A -96.2778,B 24.8866,C -2.4577,E1 24.999,E2 540.0914} C_DIS
Startdeposition()
$VEL.CP = VEL_PRINT
LIN {X 1.6127,Y -54.0776,Z 68,A -93.722,B 24.8845,C -2.4806,E1 25.0063,E2 537.4815} C_DIS
LIN {X 3.6605,Y -53.9776,Z 68,A -91.3853,B 24.8841,C -2.4847,E1 25.0129,E2 535.136} C_DIS
LIN {X 6.7265,Y -53.6823,Z 68,A -88.4674,B 24.8846,C -2.4798,E1 25.0209,E2 532.2317} C_DIS
LIN {X 9.236,Y -53.3081,Z 68,A -85.3837,B 24.8837,C -2.4895,E1 25.0295,E2 529.128} C_DIS
LIN {X 11.79,Y -52.802,Z 68,A -82.8817,B 24.8839,C -2.4869,E1 25.0363,E2 526.6354} C_DIS
LIN {X 13.3849,Y -52.4195,Z 68,A -80.7002,B 24.8829,C -2.4975,E1 25.0423,E2 524.432} C_DIS
LIN {X 16.1976,Y -51.6203,Z 68,A -77.5213,B 24.8824,C -2.5026,E1 25.0508,E2 521.2464} C_DIS
LIN {X 20.0201,Y -50.2617,Z 68,A -73.8395,B 24.8831,C -2.4957,E1 25.0604,E2 517.5887} C_DIS
LIN {X 22.4217,Y -49.2371,Z 68,A -70.5199,B 24.8816,C -2.5112,E1 25.0689,E2 514.2406} C_DIS
LIN {X 24.8072,Y -48.0794,Z 68,A -68.1549,B 24.8821,C -2.5066,E1 25.0748,E2 511.893} C_DIS
LIN {X 27.8821,Y -46.3642,Z 68,A -63.5614,B 24.8797,C -2.5313,E1 25.086,E2 507.2549} C_DIS
LIN {X 30.936,Y -44.3841,Z 68,A -60.5892,B 24.8808,C -2.5202,E1 25.0928,E2 504.3189} C_DIS
LIN {X 32.9829,Y -42.8849,Z 68,A -57.596,B 24.8796,C -2.5322,E1 25.0995,E2 501.308} C_DIS
LIN {X 34.8202,Y -41.4081,Z 68,A -55.4926,B 24.8799,C -2.5293,E1 25.104,E2 499.2195} C_DIS
LIN {X 36.2292,Y -40.1804,Z 68,A -53.4227,B 24.8793,C -2.5357,E1 25.1083,E2 497.1427} C_DIS
LIN {X 38.0212,Y -38.4886,Z 68,A -50.6195,B 24.8783,C -2.546,E1 25.114,E2 494.3268} C_DIS
LIN {X 39.7327,Y -36.7196,Z 68,A -48.2101,B 24.8781,C -2.5481,E1 25.1186,E2 491.9228} C_DIS
LIN {X 40.9753,Y -35.3284,Z 68,A -46.3973,B 24.878,C -2.5496,E1 25.1219,E2 490.1147} C_DIS
LIN {X 42.4693,Y -33.5162,Z 68,A -43.5182,B 24.8765,C -2.5645,E1 25.127,E2 487.2136} C_DIS
LIN {X 43.9891,Y -31.4952,Z 68,A -41.1862,B 24.8765,C -2.5642,E1 25.1309,E2 484.8937} C_DIS
LIN {X 45.9533,Y -28.5533,Z 68,A -36.5902,B 24.8737,C -2.5932,E1 25.1379,E2 480.2523} C_DIS
LIN {X 47.7421,Y -25.4508,Z 68,A -33.6783,B 24.8746,C -2.5847,E1 25.1418,E2 477.3756} C_DIS
LIN {X 48.9172,Y -23.1114,Z 68,A -30.4614,B 24.8728,C -2.6025,E1 25.1457,E2 474.1337} C_DIS
LIN {X 49.9718,Y -20.7336,Z 68,A -27.5228,B 24.8716,C -2.6148,E1 25.1489,E2 471.1822} C_DIS
LIN {X 51.528,Y -16.4888,Z 68,A -22.7836,B 24.8703,C -2.6284,E1 25.1532,E2 466.4376} C_DIS
LIN {X 52.5858,Y -12.7172,Z 68,A -19.5628,B 24.871,C -2.6207,E1 25.1555,E2 463.2535} C_DIS
LIN {X 53.4092,Y -8.633,Z 68,A -13.8346,B 24.8668,C -2.6637,E1 25.1584,E2 457.4571} C_DIS
LIN {X 53.9065,Y -4.5979,Z 68,A -10.5942,B 24.8678,C -2.6536,E1 25.1593,E2 454.2599} C_DIS
LIN {X 54.0395,Y -2.6067,Z 68,A -8.5531,B 24.8673,C -2.6587,E1 25.1597,E2 452.2188} C_DIS
LIN {X 54.0997,Y 0.5454,Z 68,A -4.4821,B 24.8646,C -2.6854,E1 25.1597,E2 448.1088} C_DIS
LIN {X 53.9575,Y 3.958,Z 68,A -1.7977,B 24.8655,C -2.6761,E1 25.1593,E2 445.4624} C_DIS
LIN {X 53.5347,Y 7.8139,Z 68,A 2.2884,B 24.8643,C -2.6884,E1 25.158,E2 441.3714} C_DIS
LIN {X 53.1062,Y 10.3308,Z 68,A 5.711,B 24.8618,C -2.7125,E1 25.1562,E2 437.9119} C_DIS
LIN {X 52.5399,Y 12.9051,Z 68,A 8.2153,B 24.8616,C -2.7145,E1 25.1546,E2 435.4172} C_DIS
LIN {X 51.7316,Y 15.8386,Z 68,A 11.3484,B 24.8608,C -2.7221,E1 25.1521,E2 432.284} C_DIS
LIN {X 50.9373,Y 18.2332,Z 68,A 14.0027,B 24.8601,C -2.7295,E1 25.1497,E2 429.6272} C_DIS
LIN {X 49.902,Y 20.8994,Z 68,A 16.9774,B 24.8593,C -2.737,E1 25.1466,E2 426.6514} C_DIS
LIN {X 48.6518,Y 23.6655,Z 68,A 19.8587,B 24.8591,C -2.7386,E1 25.1432,E2 423.7817} C_DIS
LIN {X 47.5928,Y 25.7276,Z 68,A 22.38,B 24.8583,C -2.7467,E1 25.14,E2 421.2546} C_DIS
LIN {X 46.5971,Y 27.49,Z 68,A 25.0396,B 24.8566,C -2.7634,E1 25.1362,E2 418.5691} C_DIS
LIN {X 44.5187,Y 30.7423,Z 68,A 29.925,B 24.8537,C -2.7908,E1 25.1285,E2 413.6431} C_DIS
LIN {X 42.3695,Y 33.6426,Z 68,A 32.6313,B 24.8553,C -2.7759,E1 25.1239,E2 410.9848} C_DIS
LIN {X 40.6968,Y 35.6477,Z 68,A 35.1486,B 24.8552,C -2.7769,E1 25.1194,E2 408.4765} C_DIS
LIN {X 39.141,Y 37.3497,Z 68,A 37.8188,B 24.8541,C -2.787,E1 25.1142,E2 405.7941} C_DIS
LIN {X 37.5345,Y 38.9633,Z 68,A 39.9151,B 24.8543,C -2.7854,E1 25.1101,E2 403.7104} C_DIS
LIN {X 35.7908,Y 40.5715,Z 68,A 42.6029,B 24.8534,C -2.794,E1 25.1045,E2 401.0131} C_DIS
LIN {X 34.0606,Y 42.034,Z 68,A 44.9138,B 24.8531,C -2.7966,E1 25.0995,E2 398.7048} C_DIS
LIN {X 32.0008,Y 43.6226,Z 68,A 47.3922,B 24.8531,C -2.7958,E1 25.094,E2 396.2374} C_DIS
LIN {X 29.0244,Y 45.6577,Z 68,A 51.329,B 24.8523,C -2.8042,E1 25.0849,E2 392.2938} C_DIS
LIN {X 26.2453,Y 47.3095,Z 68,A 55.0485,B 24.8511,C -2.815,E1 25.0759,E2 388.56} C_DIS
LIN {X 24.1995,Y 48.3878,Z 68,A 57.4201,B 24.851,C -2.8165,E1 25.07,E2 386.1913} C_DIS
LIN {X 21.9695,Y 49.4409,Z 68,A 60.3125,B 24.8501,C -2.825,E1 25.0626,E2 383.2859} C_DIS
LIN {X 19.261,Y 50.557,Z 68,A 62.7518,B 24.8511,C -2.815,E1 25.0564,E2 380.8758} C_DIS
LIN {X 17.3968,Y 51.2284,Z 68,A 65.0971,B 24.8504,C -2.8216,E1 25.0502,E2 378.5196} C_DIS
LIN {X 13.9045,Y 52.2844,Z 68,A 69.8704,B 24.8483,C -2.8419,E1 25.0372,E2 373.706} C_DIS
LIN {X 10.9038,Y 52.9914,Z 68,A 72.8784,B 24.8486,C -2.8384,E1 25.0291,E2 370.7101} C_DIS
LIN {X 6.3775,Y 53.7244,Z 68,A 77.7214,B 24.8486,C -2.8394,E1 25.0157,E2 365.8691} C_DIS
LIN {X 1.8767,Y 54.0695,Z 68,A 82.041,B 24.8495,C -2.8306,E1 25.0037,E2 361.5719} C_DIS
LIN {X -1.7257,Y 54.0741,Z 68,A 86.3116,B 24.8487,C -2.8381,E1 24.9917,E2 357.2833} C_DIS
LIN {X -4.5743,Y 53.9085,Z 68,A 89.4229,B 24.8487,C -2.8384,E1 24.9831,E2 354.17} C_DIS
LIN {X -9.4579,Y 53.2686,Z 68,A 93.5222,B 24.8511,C -2.8149,E1 24.9719,E2 350.1233} C_DIS
LIN {X -11.7556,Y 52.8089,Z 68,A 96.5827,B 24.8503,C -2.8231,E1 24.9634,E2 347.0396} C_DIS
LIN {X -14.4493,Y 52.1373,Z 68,A 99.4336,B 24.8508,C -2.8186,E1 24.9558,E2 344.1951} C_DIS
LIN {X -16.6196,Y 51.4857,Z 68,A 101.745,B 24.8512,C -2.8144,E1 24.9496,E2 341.8898} C_DIS
LIN {X -18.5854,Y 50.8091,Z 68,A 104.3235,B 24.8508,C -2.8182,E1 24.9428,E2 339.2971} C_DIS
LIN {X -21.9755,Y 49.4381,Z 68,A 107.6818,B 24.8523,C -2.804,E1 24.9342,E2 335.9651} C_DIS
LIN {X -23.9098,Y 48.5316,Z 68,A 110.3048,B 24.852,C -2.8066,E1 24.9276,E2 333.329} C_DIS
LIN {X -26.2753,Y 47.2928,Z 68,A 112.9974,B 24.8528,C -2.7996,E1 24.921,E2 330.6454} C_DIS
LIN {X -28.8535,Y 45.7658,Z 68,A 116.5799,B 24.8526,C -2.8008,E1 24.9124,E2 327.0491} C_DIS
LIN {X -31.261,Y 44.1562,Z 68,A 119.6385,B 24.8533,C -2.7947,E1 24.9054,E2 323.9948} C_DIS
LIN {X -34.1741,Y 41.9418,Z 68,A 123.3272,B 24.8545,C -2.7835,E1 24.8973,E2 320.3192} C_DIS
LIN {X -36.5182,Y 39.9175,Z 68,A 126.3652,B 24.8557,C -2.7722,E1 24.891,E2 317.2961} C_DIS
LIN {X -37.8294,Y 38.6775,Z 68,A 128.6691,B 24.8554,C -2.7741,E1 24.8864,E2 314.978} C_DIS
LIN {X -40.0958,Y 36.3229,Z 68,A 131.8306,B 24.8568,C -2.7608,E1 24.8804,E2 311.8344} C_DIS
LIN {X -41.4152,Y 34.8116,Z 68,A 134.7408,B 24.8561,C -2.7682,E1 24.8751,E2 308.8934} C_DIS
LIN {X -44.3681,Y 30.9591,Z 68,A 139.5128,B 24.8581,C -2.7486,E1 24.8672,E2 304.1451} C_DIS
LIN {X -45.7574,Y 28.8669,Z 68,A 142.2053,B 24.8588,C -2.7418,E1 24.8632,E2 301.4553} C_DIS
LIN {X -47.5639,Y 25.7807,Z 68,A 145.5782,B 24.8606,C -2.7245,E1 24.8585,E2 298.1061} C_DIS
LIN {X -49.0757,Y 22.7718,Z 68,A 149.6099,B 24.8609,C -2.7214,E1 24.8536,E2 294.0599} C_DIS
LIN {X -50.3217,Y 19.8675,Z 68,A 152.8399,B 24.8621,C -2.7096,E1 24.8502,E2 290.8402} C_DIS
LIN {X -51.3188,Y 17.1286,Z 68,A 155.8729,B 24.8632,C -2.6994,E1 24.8474,E2 287.8144} C_DIS
LIN {X -52.171,Y 14.324,Z 68,A 158.9726,B 24.8641,C -2.6897,E1 24.845,E2 284.7198} C_DIS
Enddeposition()
END
